// TwinCAT 3 PLC project SlaveController
// ProgramVersion: 3.1.4024.0
// libraries:
//   CAA Memory, * (CAA Technical Workgroup)
//   Tc2_EtherCAT, * (Beckhoff Automation GmbH)
//   Tc2_Math, * (Beckhoff Automation GmbH)
//   Tc2_Standard, * (Beckhoff Automation GmbH)
//   Tc2_System, * (Beckhoff Automation GmbH)
//   Tc2_TcpIp, * (Beckhoff Automation GmbH)
//   Tc2_Utilities, * (Beckhoff Automation GmbH)
//   Tc3_Module, * (Beckhoff Automation GmbH)
// project tree:
//   AgiMaths/Frames/ DHTrans.TcPOU (not stored), invFrame.TcPOU (not stored), rotX.TcPOU (not stored), rotY.TcPOU (not stored), rotZ.TcPOU (not stored), transform.TcPOU (not stored)
//   AgiMaths/MatrixLib/ angAxis2Rot.TcPOU (not stored), cross.TcPOU (not stored), Det5.TcPOU (not stored), Det6.TcPOU (not stored), Det7.TcPOU (not stored), invMat6.TcPOU (not stored), invMat6Old.TcPOU (not stored), invMat3.TcPOU (not stored), invMat7.TcPOU (not stored), Mat3T.TcPOU (not stored), matAdd.TcPOU (not stored), matMultiNum.TcPOU (not stored), matMultiply.TcPOU (not stored), matMultiVec.TcPOU (not stored), matSelfAdd.TcPOU (not stored), vecSelfAdd.TcPOU (not stored), matSelfSub.TcPOU (not stored), matSub.TcPOU (not stored), matTranspose.TcPOU (not stored), rot2AngAxis.TcPOU (not stored), vecAdd.TcPOU (not stored), norm.TcPOU (not stored), normalize.TcPOU (not stored), vecSelfMultiNum.TcPOU (not stored), vecMultiNum.TcPOU (not stored), vecSelfSub.TcPOU (not stored), vecSub.TcPOU (not stored)
//   AgiMaths/ sign.TcPOU (not stored), addVec7.TcPOU (not stored), atan2.TcPOU (not stored), cot.TcPOU (not stored)
//   DUTs/ Account.TcDUT
//   DUTs/Enum/ E_ArmLightCtrlWord.TcDUT (not stored), E_CartJointState.TcTLEO (not stored), E_DriverCtrlWord.TcDUT (not stored), E_DriverOPMode.TcDUT (not stored), E_DriverStatusWord.TcDUT (not stored), E_EndoscopePosture.TcDUT (not stored), E_EndoscopeType.TcDUT (not stored), E_InstrumentType.TcDUT, E_MasterArmState.TcDUT (not stored), E_MatchedSlaveArmIdx.TcDUT (not stored), E_SetupArmState.TcDUT (not stored), E_SlaveArmState.TcDUT
//   DUTs/Structure/MasterSlaveCommunication/ ST_MasterStatus.TcDUT (not stored), ST_SlaveStatus.TcDUT
//   DUTs/Structure/ ST_CartInputDataPool.TcDUT (not stored), ST_EtherCATState.TcDUT, ST_Frame.TcDUT (not stored), ST_InstruOnChipData.TcDUT, ST_InstruStatus.TcDUT (not stored), ST_InstruTypeInfo.TcDUT (not stored), ST_SetupArmCtrlCmds.TcDUT (not stored), ST_SetupInputDataPool.TcDUT (not stored), ST_SlaveArmCtrlCmds.TcDUT, ST_SlaveInputDataPool.TcDUT
//   DUTs/Structure/TasksCommunication/ ST_CartJointData.TcDUT (not stored), ST_CartMotorInput.TcDUT (not stored), ST_CartMotorOutput.TcDUT (not stored), ST_CartStatus.TcDUT (not stored), ST_CartUIData.TcDUT (not stored), ST_MasterJointData.TcDUT (not stored), ST_MotorInputs.TcDUT (not stored), ST_MotorOutputs.TcDUT (not stored), ST_SafetyData.TcDUT, ST_SetupJointData.TcDUT (not stored), ST_SetupStatus.TcDUT, ST_SlaveDynaData.TcDUT (not stored), ST_SlaveJointData.TcDUT (not stored), ST_SlaveUIData.TcDUT (not stored)
//   DUTs/Structure/UICommunication/ ST_cartOperation.TcDUT, ST_instruInfomation.TcDUT, ST_robotStateMachine.TcDUT, ST_uiControl.TcDUT
//   DUTs/Type/ Mat34.TcDUT (not stored), Mat35.TcDUT (not stored), Mat37.TcDUT (not stored), Mat3d.TcDUT (not stored), Mat43.TcDUT (not stored), Mat45.TcDUT, Mat4d.TcDUT (not stored), Mat53.TcDUT (not stored), Mat5d.TcDUT (not stored), Mat67.TcDUT (not stored), Mat6d.TcDUT (not stored), Mat76.TcDUT (not stored), Mat7d.TcDUT (not stored), Vec13d.TcDUT, Vec13di.TcDUT, Vec2i.TcDUT (not stored), Vec3i.TcDUT, Vec3d.TcDUT (not stored), Vec4b.TcDUT (not stored), Vec4d.TcDUT (not stored), Vec4i.TcDUT (not stored), Vec5b.TcDUT (not stored), Vec5d.TcDUT (not stored), Vec5i.TcDUT (not stored), Vec6d.TcDUT (not stored), Vec6i.TcDUT (not stored), Vec7d.TcDUT (not stored), Vec7i.TcDUT (not stored), Vec8b.TcDUT, Vec8d.TcDUT (not stored), Vec8di.TcDUT, Vec8i.TcDUT (not stored)
//   FBs_Auxiliary/ FB_cartJntDisenableDetect.TcPOU (not stored), FB_cartJntEnableDetect.TcPOU (not stored), FB_initMotorPID.TcPOU, FB_InstruNearDetect.TcPOU (not stored), FB_IOCheck.TcPOU (not stored), FB_IOToggleCheck.TcPOU (not stored), FB_rotaButtonDetect.TcPOU (not stored), FB_setupAdjustDetect.TcPOU (not stored), FB_setupJnt5AdjustDetect.TcPOU (not stored), FB_masterConnectionCheck.TcPOU (not stored), FB_Timer.TcPOU, FB_trocarDetect.TcPOU (not stored), FB_PanelDetect.TcPOU, FB_InstrumentDetect.TcPOU, FB_AdjustDetect.TcPOU (not stored)
//   FBs_BasicControllers/ FB_dither.TcPOU (not stored), FB_BasicInstruControl.TcPOU, FBMacroJntControl.TcPOU (not stored), FB_UltrosonicKnifeControl.TcPOU, FB_PID.TcPOU (not stored)
//   FBs_Robots/ FB_Instrument.TcPOU, FB_JointBase.TcPOU (not stored), FB_SlaveCart.TcPOU (not stored), FB_SlaveJoint.TcPOU, FB_SlaveArm.TcPOU, FB_SlaveRobot.TcPOU
//   FBs_SlaveControllers/ FB_SlaveCtrlDisable.TcPOU (not stored), FB_SlaveCtrlInstruCali.TcPOU, FB_SlaveCtrlInstruInvasion.TcPOU (not stored), FB_SlaveCtrlInstruEndoscopeTest.TcPOU, FB_SlaveCtrlInstruRetract.TcPOU (not stored), FB_SlaveCtrlInstruManualTest.TcPOU, FB_SlaveCtrlMountInstru.TcPOU, FB_SlaveCtrlPerformance.TcPOU (not stored), FB_SlaveCtrlPowerBoxCalibration.TcPOU, FB_SlaveCtrlScopeToggle.TcPOU (not stored), FB_SlaveCtrlStop.TcPOU, FB_SlaveCtrlTest.TcPOU, FB_SlaveCtrlPackage.TcPOU (not stored), FB_SlaveCtrlEndoscope.TcPOU (not stored), FB_SlaveCtrlCart.TcPOU (not stored), FB_SlaveCtrlScopeReady.TcPOU (not stored), FB_SlaveCtrlSelfCheck.TcPOU (not stored), FB_SlaveCtrlError.TcPOU, FB_SlaveCtrlInstruReady.TcPOU (not stored), FB_SlaveCtrlMasterSlave.TcPOU, FB_SlaveCtrlAdjust.TcPOU, FB_SlaveCtrlMountPanel.TcPOU, FB_SlaveCtrlPanelReady.TcPOU (unreadable), FB_SlaveCtrlGraCali.TcPOU (not stored), FB_SlaveCtrlInstruAutoTest.TcPOU, FB_SlaveCtrlInstruVerify.TcPOU, FB_SlaveCtrlFrictionTest.TcPOU, FB_SlaveCtrMotorGoHome.TcPOU, FB_SlaveCtrlInit.TcPOU, FB_SlaveCtrlStandBy.TcPOU (unreadable), FB_SlaveArmCtrlBase.TcPOU, I_SlaveArmCtrl.TcIO (not stored)
//   FBs_TrajectoryPlanning/ FB_BasicDoubleS.TcPOU (not stored), FB_trajBase.TcPOU (not stored), FB_TrajMoveJ.TcPOU (not stored), FB_setupTrajMoveJ.TcPOU (not stored), linear_trajectory_with_quintic_polynomial_blends.TcPOU (not stored), quintic_spline_curve.TcPOU (not stored), Quintic_spline_curve_factor.TcPOU (not stored), TrapezoIDal_velocity_trajectory.TcPOU (not stored)
//   FBs_TrajectoryPlanning/OTG/ FB_secOrdTrajFilter.TcPOU (not stored), FB_thirdOrdTrajFilter.TcPOU (not stored)
//   FBs_Filters/ FB_LowPassFilter.TcPOU (not stored)
//   GVLs/ GVL_InstruTestUIVars.TcGVL, GVL_MathDefine.TcGVL, GVL_MES.TcGVL, GVL_SafetyParameters.TcGVL (not stored), GVL_SystemParameters.TcGVL
//   GVLs/Instrument/ GVL_InstruCtrlParams.TcGVL, GVL_InstruTypeDefine.TcGVL
//   GVLs/SlaveArms/ GVL_SlaveArmDynamics.TcGVL, GVL_SlaveArmKinematic.TcGVL (not stored), GVL_SlaveControlParameters.TcGVL, GVL_SlaveJointEncoderCaliData.TcGVL, GVL_SlaveMotorParameters.TcGVL
//   Mains/ SlaveArmControl.TcPOU
//   / RecipeManager.TcRMO (not stored), TaskSlaveArmControl.TcTTO (not stored)
//   SafetyCheck/ ASSERT.TcPOU (not stored), FB_CartCheck.TcPOU (not stored), Fb_ErrRecord.TcPOU (not stored), FB_EtherCATCheck.TcPOU (not stored), Fb_SafetyCheck.TcPOU (not stored), FB_SetupArmCheck.TcPOU (not stored), FB_SlaveArmCheck.TcPOU (not stored), FB_Writer.TcPOU (not stored)
//   SafetyCheck/ErrRecord/ CarErrInputVariable.TcDUT (not stored), checkDelay.TcDUT (not stored), checkDelayTime.TcDUT (not stored), checkInputVariable.TcDUT (not stored), checkPermit.TcDUT (not stored), monitorThreshold.TcDUT (not stored), monitorThreshold_1.TcDUT (not stored), PromptMessage.TcDUT (not stored), ST_Buffer.TcDUT (not stored), T_Buffer.TcDUT (not stored)
//   Sandbox/ FB_SlaveCtrlInstruAutoTest_bak.TcPOU, FB_SlaveCtrlInstruVerify_bak.TcPOU, FB_SlaveCtrlMasterSlave_backup.TcPOU
// real-time tasks:
//   TASK TaskSlaveArmControl: cycle T#250us, priority 1, ADS port 350
// I/O:
//   DEVICE Device 3 (EtherCAT), AmsNetId 192.168.2.195.4.1
//     Box 1 (AX58200_MotorControl) [AX58200_MotorControl_V1001]
//     Box 2 (AX58200_MotorControl) [AX58200_MotorControl_V1001]
// variable links:
//   SlaveController/SlaveController Instance <-> Device 3 (EtherCAT)/Box 1 (AX58200_MotorControl)
//     TaskSlaveArmControl Inputs/SlaveArmControl.m_slaveRobot.m_slaveArms[1].m_joints[4].m_motorInputs/m_current <-> TxPdoMappingCsv/Torque actual value for axis2
//     TaskSlaveArmControl Inputs/SlaveArmControl.m_slaveRobot.m_slaveArms[1].m_joints[5].m_motorInputs/m_current <-> TxPdoMappingCsv/Torque actual value for axis3
//     TaskSlaveArmControl Inputs/SlaveArmControl.m_slaveRobot.m_slaveArms[1].m_joints[4].m_motorInputs/m_linkEncoder <-> TxPdoMappingCsv/ENC for axis2
//     TaskSlaveArmControl Inputs/SlaveArmControl.m_slaveRobot.m_slaveArms[1].m_joints[5].m_motorInputs/m_linkEncoder <-> TxPdoMappingCsv/ENC for axis3
//     TaskSlaveArmControl Inputs/SlaveArmControl.m_slaveRobot.m_slaveArms[1].m_joints[4].m_motorInputs/m_motorEncoder <-> TxPdoMappingCsv/Position actual value for axis2
//     TaskSlaveArmControl Inputs/SlaveArmControl.m_slaveRobot.m_slaveArms[1].m_joints[5].m_motorInputs/m_motorEncoder <-> TxPdoMappingCsv/Position actual value for axis3
//     TaskSlaveArmControl Inputs/SlaveArmControl.m_slaveRobot.m_slaveArms[1].m_joints[4].m_motorInputs/m_statusWord <-> TxPdoMappingCsv/Statusword
//     TaskSlaveArmControl Inputs/SlaveArmControl.m_slaveRobot.m_slaveArms[1].m_joints[5].m_motorInputs/m_statusWord <-> TxPdoMappingCsv/Statusword
//     TaskSlaveArmControl Inputs/SlaveArmControl.m_slaveRobot.m_slaveArms[1].m_panelInstrumentOnIO <-> TxPdoMappingCsv/Digital input
//     TaskSlaveArmControl Outputs/SlaveArmControl.m_slaveRobot.m_slaveArms[1].m_joints[4].m_motorOutputs/m_cmdCurrent <-> RxPdoMappingCsv/Target torque for axis2
//     TaskSlaveArmControl Outputs/SlaveArmControl.m_slaveRobot.m_slaveArms[1].m_joints[5].m_motorOutputs/m_cmdCurrent <-> RxPdoMappingCsv/Target torque for axis3
//     TaskSlaveArmControl Outputs/SlaveArmControl.m_slaveRobot.m_slaveArms[1].m_joints[4].m_motorOutputs/m_cmdMotorEncoder <-> RxPdoMappingCsv/Target position for axis2
//     TaskSlaveArmControl Outputs/SlaveArmControl.m_slaveRobot.m_slaveArms[1].m_joints[5].m_motorOutputs/m_cmdMotorEncoder <-> RxPdoMappingCsv/Target position for axis3
//     TaskSlaveArmControl Outputs/SlaveArmControl.m_slaveRobot.m_slaveArms[1].m_joints[4].m_motorOutputs/m_controlWord <-> RxPdoMappingCsv/Controlword
//     TaskSlaveArmControl Outputs/SlaveArmControl.m_slaveRobot.m_slaveArms[1].m_joints[4].m_motorOutputs/m_opMode <-> RxPdoMappingCsv/Modes of operation
//   SlaveController/SlaveController Instance <-> Device 3 (EtherCAT)/Box 2 (AX58200_MotorControl)
//     TaskSlaveArmControl Inputs/SlaveArmControl.m_slaveRobot.m_slaveArms[1].m_joints[6].m_motorInputs/m_current <-> TxPdoMappingCsv/Torque actual value for axis2
//     TaskSlaveArmControl Inputs/SlaveArmControl.m_slaveRobot.m_slaveArms[1].m_joints[7].m_motorInputs/m_current <-> TxPdoMappingCsv/Torque actual value for axis3
//     TaskSlaveArmControl Inputs/SlaveArmControl.m_slaveRobot.m_slaveArms[1].m_joints[6].m_motorInputs/m_linkEncoder <-> TxPdoMappingCsv/ENC for axis2
//     TaskSlaveArmControl Inputs/SlaveArmControl.m_slaveRobot.m_slaveArms[1].m_joints[7].m_motorInputs/m_linkEncoder <-> TxPdoMappingCsv/ENC for axis3
//     TaskSlaveArmControl Inputs/SlaveArmControl.m_slaveRobot.m_slaveArms[1].m_joints[6].m_motorInputs/m_motorEncoder <-> TxPdoMappingCsv/Position actual value for axis2
//     TaskSlaveArmControl Inputs/SlaveArmControl.m_slaveRobot.m_slaveArms[1].m_joints[7].m_motorInputs/m_motorEncoder <-> TxPdoMappingCsv/Position actual value for axis3
//     TaskSlaveArmControl Inputs/SlaveArmControl.m_slaveRobot.m_slaveArms[1].m_joints[6].m_motorInputs/m_statusWord <-> TxPdoMappingCsv/Statusword
//     TaskSlaveArmControl Inputs/SlaveArmControl.m_slaveRobot.m_slaveArms[1].m_joints[7].m_motorInputs/m_statusWord <-> TxPdoMappingCsv/Statusword
//     TaskSlaveArmControl Inputs/SlaveArmControl.m_slaveRobot.m_slaveArms[1].m_joints[8].m_motorInputs/m_statusWord <-> TxPdoMappingCsv/Statusword
//     TaskSlaveArmControl Inputs/SlaveArmControl.m_slaveRobot.m_slaveArms[1].m_joints[8].m_motorInputs/m_current <-> TxPdoMappingCsv/Torque actual value
//     TaskSlaveArmControl Inputs/SlaveArmControl.m_slaveRobot.m_slaveArms[1].m_joints[8].m_motorInputs/m_linkEncoder <-> TxPdoMappingCsv/ENC
//     TaskSlaveArmControl Inputs/SlaveArmControl.m_slaveRobot.m_slaveArms[1].m_joints[8].m_motorInputs/m_motorEncoder <-> TxPdoMappingCsv/Position actual value
//     TaskSlaveArmControl Outputs/SlaveArmControl.m_slaveRobot.m_slaveArms[1].m_joints[6].m_motorOutputs/m_cmdCurrent <-> RxPdoMappingCsv/Target torque for axis2
//     TaskSlaveArmControl Outputs/SlaveArmControl.m_slaveRobot.m_slaveArms[1].m_joints[7].m_motorOutputs/m_cmdCurrent <-> RxPdoMappingCsv/Target torque for axis3
//     TaskSlaveArmControl Outputs/SlaveArmControl.m_slaveRobot.m_slaveArms[1].m_joints[6].m_motorOutputs/m_cmdMotorEncoder <-> RxPdoMappingCsv/Target position for axis2
//     TaskSlaveArmControl Outputs/SlaveArmControl.m_slaveRobot.m_slaveArms[1].m_joints[7].m_motorOutputs/m_cmdMotorEncoder <-> RxPdoMappingCsv/Target position for axis3
//     TaskSlaveArmControl Outputs/SlaveArmControl.m_slaveRobot.m_slaveArms[1].m_joints[6].m_motorOutputs/m_controlWord <-> RxPdoMappingCsv/Controlword
//     TaskSlaveArmControl Outputs/SlaveArmControl.m_slaveRobot.m_slaveArms[1].m_joints[6].m_motorOutputs/m_opMode <-> RxPdoMappingCsv/Modes of operation
//     TaskSlaveArmControl Outputs/SlaveArmControl.m_slaveRobot.m_slaveArms[1].m_joints[8].m_motorOutputs/m_cmdCurrent <-> RxPdoMappingCsv/Target torque
//     TaskSlaveArmControl Outputs/SlaveArmControl.m_slaveRobot.m_slaveArms[1].m_joints[8].m_motorOutputs/m_cmdMotorEncoder <-> RxPdoMappingCsv/Target position

// ---- DUTs/Account.TcDUT
TYPE Account :
STRUCT
	logOn:BOOL;
	logOut:BOOL;
	autoLogOut:BOOL;
	register:BOOL;//注册
	actualAccountNumber:STRING;
	actualPassWord:STRING;
	actualPermission:USINT;//权限 0 无登录 1 管理 2 研发 3 质量 4 生产
	actualWorkNum:UDINT;
	actualName:STRING;
	registerAccountNumber:STRING;
	registerPassWord:STRING;
	registerPermission:USINT;
	registerWorkNum:UDINT;
	registerName:STRING;
	prompt:STRING;//提示
	memoryAccountNumber:ARRAY [0..50] OF STRING; //注册账号
	memoryPassWord:ARRAY [0..50] OF STRING; //注册账密码
	memoryPermission:ARRAY [0..50] OF USINT; //注册账权限
	memoryWorkNum:ARRAY [0..50] OF UDINT;//注册账工号
	memoryName:ARRAY [0..50] OF STRING; //注册账姓名
	memoryTime:ARRAY [0..50] OF STRING; //注册时间
	memoryDisable:ARRAY [0..50] OF BOOL;//使能
END_STRUCT
END_TYPE

// ---- DUTs/Enum/E_InstrumentType.TcDUT
TYPE E_InstrumentType :
(
	InstruType_UNKNOWM := 0,
	InstruType_CadiereForceps :=7,
	InstruType_NeedleDriver :=8,
	InstruType_MegaSCNeedleDriver :=9,// mega suture-cut needle driver
	InstruType_SCNeedleDriver :=10, // suture-cut needle driver
	InstruType_RoundTipScissors :=11,
	InstruType_ProGraspForceps :=12,
	InstruType_MarylandForceps :=13, // Maryland bipolar forceps
	InstruType_FenestratedForceps :=14, // Fnestrated bipolar forceps
	InstruType_CurvedScissors :=15, // monopolar curved scissors
	InstruType_CauteryHook :=16,
	InstruType_CauterySpatula :=17,
	InstruType_Endoscope := 20,
	InstruType_NewEndoscope := 31,
	InstruType_UltrasoundKnifeS :=42,
	InstruType_UltrasoundKnifeU :=43,
	InstruType_TipUpFenestratedGrasper :=44,
	InstruType_MegaNeedleDriver :=45,
	InstruType_DeBakeyForceps :=46,
	InstruType_BlackDiamondForceps :=47,
	InstruType_PottsScissors :=48,
	InstruType_CurvedBipolarDissector :=49,
	InstruType_MicroBipolarForceps :=50,
	InstruType_ForceBipolar :=51,
	InstruType_MicroCauteryHook :=52,
	InstruType_CENewEndoscope := 320
);
END_TYPE

// ---- DUTs/Enum/E_SlaveArmState.TcDUT
TYPE E_SlaveArmState :
(
	SlaveArmState_Error := 1,
	SlaveArmState_Init :=2,
	SlaveArmState_SelfCheck :=3,
	SlaveArmState_Standby :=4,
	SlaveArmState_MountPanel:=5,
	SlaveArmState_PanelReady :=6,
	SlaveArmState_MountInstru :=7,
	SlaveArmState_InstruReady :=8,
	SlaveArmState_MasterSlave :=9,
	SlaveArmState_ScopeReady :=10,
	SlaveArmState_EndoScope :=11,
	SlaveArmState_Adjust :=12,
	SlaveArmState_Package :=13,
	SlaveArmState_Cart := 14,
	SlaveArmState_GravityCali := 15,
	SlaveArmState_Test := 16,
	SlaveArmState_InstruRetract :=17,
	SlaveArmState_InstruInvasion :=18,
	SlaveArmState_Disable := 19,
	SlaveArmState_InstruCali := 20,
	SlaveArmState_ScopeToggle :=21,
	SlaveArmState_Performance:=22,
	SlaveArmState_Stop :=23,
	SlaveArmState_InstruAutoTest :=24,
	SlaveArmState_InstruManualTest :=25,
	SlaveArmState_InstruVerify :=26,
	SlaveArmState_MotorGoHome:= 27,
	SlaveArmState_PowerBoxCalibration:= 28,
	SlaveArmState_EndoscopeTest:= 29,
	SlaveArmState_FrictionTest:= 30,
	
	SlaveArmState_Jnt5Rotate:=31,
	SlaveArmState_totalNum :=SlaveArmState_Jnt5Rotate
);
END_TYPE

// ---- DUTs/Structure/MasterSlaveCommunication/ST_SlaveStatus.TcDUT
// Output from slave arm control task, including arm status and cartesian data
// Input to safety task and Master controller
TYPE ST_SlaveStatus :
STRUCT
	
	// state machine
	m_armState:ARRAY[1..g_sArmNum] OF E_SlaveArmState:=[g_sArmNum(SlaveArmState_Error)];
	
	// self-check pass flag
	m_selfCheckPass :ARRAY[1..g_sArmNum] OF BOOL :=[g_sArmNum(False)];
	
	// instrument info
	m_instruStauts :ARRAY[1..g_sArmNum] OF ST_InstruStatus;
	
	// flag if endoscope is mounted
	m_endoscopeMounted :BOOL := FALSE;
	
	// endoscope pose in cart coordinate
	m_endoscopePose : ST_Frame;
	
	// command arm pose in slave arm coordinate
	m_cmdArmPose:ARRAY[1..g_sArmNum] OF ST_Frame;
	
	// current arm pose in slave arm coordinate
	m_curArmPose:ARRAY[1..g_sArmNum] OF ST_Frame;
	
	// simulation arm pose in slave arm coordinate
	m_simArmPose:ARRAY[1..g_sArmNum] OF ST_Frame;
	
	// master slave pose error [position, angle*axis] in endoscope coordinate
	m_masterSlavePoseError :ARRAY[1..g_sArmNum] OF Vec6d; 

	//read instrument information error ID
	m_instruReadErrId : ARRAY[1..g_sArmNum] OF INT;
	
	//instrument install status
	m_instruInstallStatus : ARRAY[1..g_sArmNum] OF BOOL;
	
	//instrument clamp error Id 
	m_instruClampErrId : ARRAY[1..g_sArmNum] OF UINT;
	
	//panel install status
	m_panelInstallStatus : ARRAY[1..g_sArmNum] OF BOOL;
	
	//panel clamp error ID
	m_panelClampErrId : ARRAY[1..g_sArmNum] OF UINT;
	
	//trocar install status 
	m_trocarOnFlag : ARRAY[1..g_sArmNum] OF BOOL;

	// flag if master are connected
	m_masterOnLine :BOOL ;
	
	// slave robot stop button trigger 
	m_slaveStopButton : BOOL;
END_STRUCT
END_TYPE

// ---- DUTs/Structure/ST_EtherCATState.TcDUT
TYPE ST_EtherCATState :
STRUCT
	EtherCATState : BOOL;
	CRCPortA :UDINT;
	CRCPortB :UDINT;
	CRCPortC :UDINT;
END_STRUCT
END_TYPE

// ---- DUTs/Structure/ST_InstruOnChipData.TcDUT
TYPE ST_InstruOnChipData :
STRUCT

	// ID
	m_InstruID: INT:=0;
	
	// series number
	m_InstruseriesNum : ULINT:=0;
	
	// current and max usage counts
	m_InstruUsageCounts :ULINT;
	m_InstrumaxUsageCounts :ULINT:=20;
	
	//Instrument Zero augular offset
	m_InstruPos:Vec5d;
	//Instrument RFID 
	m_InstruPosRFID:Vec5d;
	m_InstruIDFromRFID: INT:=0;
	m_InstruUsageCountsRFID :ULINT;
	m_InstruReadSucceedRFID:BOOL;
	m_InstruseriesNumRFID : ULINT:=0;
	//Instrument state
	m_InstruReadSucceed:BOOL;
	
	//Instrument Clamp Error
	m_Error:BOOL;
	m_ErrorID:INT;//1器械类型错误、2器械使用次数超限、3两个内窥镜
	
	m_InstruPurpose :ULINT;
	m_InstruPurposeTime :ULINT;
END_STRUCT
END_TYPE

// ---- DUTs/Structure/ST_SlaveArmCtrlCmds.TcDUT
TYPE ST_SlaveArmCtrlCmds :
STRUCT
	// arm control data
	// NOTE: simulated joint position is usd for kinematic controller 
	//		while command joint position is used for real robot controller
	// 		They are identical for the most time, but in some cases, simulated position is filted to get command one 
	m_jntEnableFlag : Vec8i;
	m_jntOPMode : Vec8i;
	m_simJntPos : Vec8d;
	m_cmdJntPos : VEC8d;
	m_cmdJntVel : VEC8d;
	m_cmdJntAcc : VEC8d:=g_zeroVec8d;
	m_cmdJntTrq : VEC8d:=g_zeroVec8d;
	m_cmdCartPose : ST_Frame;
	m_cmdCartTwist : Vec6d;
	m_FFJntTrq :Vec8d:=g_zeroVec8d;
	
END_STRUCT
END_TYPE

// ---- DUTs/Structure/ST_SlaveInputDataPool.TcDUT
// Struct contains all data from other tasks and controller used for slave control
TYPE ST_SlaveInputDataPool :
STRUCT
		
	// UI information, import from UI controller
	m_UIData :ST_SlaveUIData;
	
	// safety information, import from safety check task
	m_safetyData : ST_SafetyData;
	
	// cart information, import from other task
	m_cartStatus :ST_CartStatus;
	
	// master robot status, copy from MSCommu_MasterStatus
	m_masterStatus :ST_MasterStatus;
	
	// setup arms infromation;
	m_setupStatus : ST_SetupStatus;
	
	// slave dynamic data
	m_slaveDynaData : ST_SlaveDynaData;
	
END_STRUCT
END_TYPE

// ---- DUTs/Structure/TasksCommunication/ST_SafetyData.TcDUT
// Output from safety check task
// Input to master arm control task
TYPE ST_SafetyData :
STRUCT
	m_slaveErrFlag :ARRAY[1..g_sArmNum] OF BOOL :=[g_sArmNum(FALSE)];
	m_setupErrFlag :ARRAY[1..g_sArmNum] OF BOOL :=[g_sArmNum(FALSE)];
	m_cartErrFlag :BOOL :=FALSE;
	m_cartSteadyFootErr :BOOL;
	m_cartWheelErr :BOOL;
	m_cartStandColumnErr :BOOL;
	m_cartAdjustErr :BOOL;
	m_cartOverhangErr :BOOL;
END_STRUCT
END_TYPE

// ---- DUTs/Structure/TasksCommunication/ST_SetupStatus.TcDUT
TYPE ST_SetupStatus :
STRUCT
	// state machine
	m_armState:ARRAY[1..g_sArmNum] OF E_SetupArmState:=[g_sArmNum(SetupArmState_Error)];
	
	// current pose of set arm distal end
	m_curEndPose:ARRAY[1..g_sArmNum] OF ST_Frame;
	
	// position of remote center point
	m_rcPos :ARRAY[1..g_sArmNum] OF Vec3d;
END_STRUCT
END_TYPE

// ---- DUTs/Structure/UICommunication/ST_cartOperation.TcDUT
TYPE ST_cartOperation :
STRUCT
	//sterile state ,  0 : unfinshed  , 1 : complete
	m_setupSterileStateArm1 : UINT;
	m_setupSterileStateArm2 : UINT;
	m_setupSterileStateArm3 : UINT;
	m_setupSterileStateArm4 : UINT;
	
	//draping adjust state , 0 : unfinshed  , 1 : finshed
	m_drapingAdjustState : UINT;

	//sterile install state , 0 : unfinshed  , 1 : finshed
	m_setupSterileState : UINT;

	//docking adjust state , 0 : unfinshed  , 1 : finshed
	m_dockingAdjustState : UINT;
	
	//cart in the sterile area 
	m_cartInSterileState : UINT;
	
	//scope installed , 0 : unfinshed  , 1 : finshed
	m_scopeInstalled :UINT;
	
	//robot in surgical allowed , scope installed and an arm mounted instrument
	m_inSurgicalAllowed : UINT;
	
	//arm storage completed
	m_armStorageCompleted : UINT;
END_STRUCT
END_TYPE

// ---- DUTs/Structure/UICommunication/ST_instruInfomation.TcDUT
TYPE ST_instruInfomation :
STRUCT
	//instrument is ready
	m_instruIsConnected : BOOL;
	
	//new instrument  true
	m_newInstrument : BOOL;
	
	//instrument arm in master-slave
	m_instruInMasterSlave : BOOL;
	
	//master send  pedal active
	m_pedalHover : BOOL;
	
	//0 : Passive instrument , 1 : unipolar instrument , 2 : bipolar instrument, 3 : ultrasound knife, 4 : endoscope
	m_instruType : UINT;
	
	//master send  pedal hover
	m_pedalActive : UINT;
	
	//arm id
	m_armId : UINT;
	m_instruID : UINT;
	
	//instrument total number
	m_instruTotalLife : UINT := 100;
	
	//instrument use life (ui write)
	m_useLifeUi : UINT;

	//instrument  use life (plc write)
	m_useLifeplc : UINT;
	
	//instrument serial number
	m_instruSerialNum : LINT;
	
	m_instruPosX : REAL;
	m_instruPosY : REAL;
	m_instruPosZ : REAL;

	//instrument English name 
	m_nameEn : STRING;
	
	//instrument Chinese name 
	m_nameCh : WSTRING;
	
END_STRUCT
END_TYPE

// ---- DUTs/Structure/UICommunication/ST_robotStateMachine.TcDUT
TYPE ST_robotStateMachine :
STRUCT
	m_stateMachineCart : INT;
	m_stateMachineArm1 : INT;
	m_stateMachineArm2 : INT;
	m_stateMachineArm3 : INT;
	m_stateMachineArm4 : INT;

END_STRUCT
END_TYPE

// ---- DUTs/Structure/UICommunication/ST_uiControl.TcDUT
TYPE ST_uiControl :
STRUCT
	//台车自动摆位---姿态调整为建立无菌屏障时所需状态--结束后给定结束信号
	m_drapingEnable : BOOL;
	
	//台车自动摆位---姿态调整为进入无菌区时所需状态（器械对接姿态）--结束后给定结束信号
	m_dockingEnable : BOOL;
	
	//所有机械臂收纳使能
	m_packageEnable : BOOL;
	
	//通过手柄按钮，任意拖动机械臂所有关节
	m_joystickEnable : BOOL;
	
	//相机界面中的使能按钮
	m_cameraJoystickEnable : BOOL;
	
	 //限制高度调整，true:使能，false:禁止
	m_heightLimitAdjustEnable : BOOL;
END_STRUCT
END_TYPE

// ---- DUTs/Type/Mat45.TcDUT
TYPE Mat45 : ARRAY[1..4, 1..5] OF LREAL; END_TYPE

// ---- DUTs/Type/Vec13d.TcDUT
TYPE Vec13d : ARRAY[1..13] OF LREAL; END_TYPE

// ---- DUTs/Type/Vec13di.TcDUT
TYPE Vec13di : ARRAY[1..13] OF DINT; END_TYPE

// ---- DUTs/Type/Vec3i.TcDUT
TYPE Vec3i : ARRAY[1..3] OF INT; END_TYPE

// ---- DUTs/Type/Vec8b.TcDUT
TYPE Vec8b : ARRAY[1..8] OF BOOl; END_TYPE

// ---- DUTs/Type/Vec8di.TcDUT
TYPE Vec8di : ARRAY[1..8] OF DINT; END_TYPE

// ---- GVLs/GVL_InstruTestUIVars.TcGVL
{attribute 'qualified_only'}
VAR_GLOBAL
	//################ input variables from HMI ########################
	// control variable for instrument calibration
	g_instruCaliFlag :BOOL:= FALSE; // 允许标定按键，按下不反弹
	g_searchZeroPosFlag :BOOL := FALSE; // 器械找零点按键， 按下反弹
	g_writeZeroPosFlag :BOOL :=FALSE; // 器械零位写入，按下反弹
	g_newInstruSN :STRING; // 新序列号
	g_writeSNFlag :BOOL := FALSE; // 新序列号写入， 按下反弹
	
	// control variable for instrument auto test
	g_instruAutoTestFlag :BOOL :=FALSE; // 器械自动测试按键，按下不反弹
	g_instruAutoTestMode :INT :=0; //  自动测试模式 0: 器械开合 1: 器械开合加运动 ; 2: 器械加紧运动
	g_maxInstruAutoTestCycles :DINT :=0; // 最大测试次数
	g_autoTestCycles :INT :=0;
	// control variable for instrument manual test
	g_instruManualTestFlag :BOOL :=FALSE; // 器械手动测试按键，按下不反弹
	g_moveToSetPosFlag :BOOL :=FALSE; // 运动到指令位置 ，按下反弹
	g_targetRollAng :LREAL :=0; //器械回转角度
	g_targetPitchAng :LREAL :=0;//器械俯仰角度
	g_targetYawAng :LREAL :=0;//器械偏摆角度
	g_targetGripAng :LREAL :=0;//器械张开角度
	g_targetGripForceLevel:INT :=0; // 器械夹持力百分比
	g_gripperOpenFlag :BOOL :=FALSE; // 命令器械张开按键, 按下反弹
	g_gripperCloseFlag :BOOL :=FALSE; // 命令器械闭合按键, 按下反弹
	g_maxGripForceFlag :BOOL :=FALSE;// 命令器械最大加紧力按键, 按下反弹
	g_forceBipolarMode : BOOL := FALSE;
	g_forceBipolarModeAllowed : BOOL := FALSE;
	
	// control variable for instrument verify
	g_instruVerifyFlag :BOOL :=FALSE; // 器械验证按键，按下不反弹
	g_instruVerifyLastStepFlag :BOOL:=FALSE; // 下一步按键， 按下反弹
	g_instruVerifyNextStepFlag :BOOL :=FALSE; // 上一步按键，按下反弹
	
	//friction test
	g_instruFrictionTestAllowed : BOOL;
	g_instruFrictionTest : BOOL;
	
	//################ output variables  HMI ########################
	g_curInstruJntPos :Vec5d;   // 当前器械角度位置
	g_curInstruJntCurrent:Vec5d; // 当前关节电流
	g_curInstruDHPos :Vec3d; // DH 角度
	g_curGripAng:LREAL; // 当前张开角度
	g_instruZeroPos :Vec5d; // 当前零位
	g_instruSN :STRING; // 当前序列号
	g_maxGripAng:LREAL:=45; // 当前张开角度
	// 读取器械信息
	g_readInstruInformation: BOOL;
	// 信息校验通过
	g_informationVerificationPassed: BOOL;
	// 电机使能
	g_powerOn: BOOL;
	// 电机使能状态
	g_enabled: BOOL;
	// 卡接隔离板
	g_snappingSeparator: BOOL;
	// 电机停止
	g_motorStops: BOOL;
	// 器械卡接找点
	g_instrumentSnapping: BOOL;
	// 器械自动卡接
	g_instrumentAutoSnapping: BOOL;
	// 器械卡接停止
	g_instrumentSnappingStop: BOOL;
	// 位置写入芯片
	g_positionWritingChip: BOOL;
	// 位置数据写入
	g_writeENC2PosData: LREAL;
	// 读取器械信息状态
	g_readInstruinformationFlag: BOOL;
	// 读取到的SN码
	g_readSNNum: ULINT;
	// 器械使用次数
	g_instruNumberOfUses: UINT;
	// 器械总使用次数
	g_instruNumberOfAllUses: UINT;
	// 增加使用次数
	g_incInstruNumOfUses: BOOL;
	// 清除使用次数
	g_clearInstruNumOfUses: BOOL;
	// 位置从芯片读取
	g_readENC2PosData: BOOL;
	// 写入器械中的SN码
	g_writeSNNum: ULINT;
	// 写入SN码
	g_writeInstruSN: BOOL;
	// 写入器械用途
	g_writeInstruPurpose: BOOL;
	// 写入器械的用途
	g_writePurposeNum: UINT;
	// 修改额定电流
	g_modifyRatedCurrent: BOOL;
	// 目标额定电流
	g_targetRatedCurrent: LREAL;
	// 实际额定电流
	g_actualRatedCurrent: ARRAY[1..g_sJntNum] OF LREAL := [8(800)];
	// 动力盒标定状态
	g_powerBoxCalibrationFlag: BOOL := TRUE;
	// 动力盒标定
	g_powerBoxCalibration: BOOL;
	// 动力盒回零位
	g_goHome: BOOL;
	
	// 读取器械用途
	g_readInstruPurpose: UINT;
	// 读取器械的用途
	g_readPurposeTime: UINT;	
	g_instruNameCN : WSTRING := " ";
	
	// 清除壳体次数
	g_jnt5RotateFlag:BOOL:=FALSE;
END_VAR
VAR_GLOBAL RETAIN PERSISTENT
	// 动力盒零位已校准
	g_powerBoxCalibrationed: BOOL;
	// 动力盒零位
	g_powerBoxCalibrationPos: ARRAY [1..g_sArmNum, 1..g_sJntNum] OF DINT;
	// 账户
	g_account: Account := (memoryAccountNumber := ['admin', 50('')], memoryPassWord := ['yfAGIBOT2025', 50('')], memoryPermission := [1, 50(0)], memoryWorkNum := [1, 50(0)], memoryName := ['admin', 50('')]);
END_VAR
VAR_GLOBAL
	// 动力盒零位状态
	g_beHomed: BOOL;
	// 后台启用角度补偿
	g_enableBackendCompensation: BOOL;
	// 研发启用角度补偿
	g_enableRDCompensation: BOOL;
	// DH补偿角度
	g_compensationAngleDH: Vec3d;
	// DH补偿角度内部
	g_compensationAngleBackendDH: Vec3d;
	// 俯仰
	g_pitchAngularVel: LREAL;
	// 偏摆/开合
	g_deviationAngularVel: LREAL;
	// 旋转
	g_rotationAngularVel: LREAL;
	// 俯仰加速度
	g_pitchAngularAcc: LREAL;
	// 偏摆/开合加速度
	g_deviationAngularAcc: LREAL;
	// 旋转加速度
	g_rotationAngularAcc: LREAL;
	// 俯仰目标电流
	g_pitchTargetCurrent: LREAL;
	// 偏摆/开合目标电流
	g_deviationTargetCurrent: LREAL;
	// 旋转目标电流
	g_rotationTargetCurrent: LREAL;
	// 俯仰当前电流
	g_pitchActualCurrent: LREAL;
	// 偏摆/开合当前电流
	g_deviationActualCurrent: LREAL;
	// 旋转当前电流
	g_rotationActualCurrent: LREAL;
	// 当前状态集
	g_stateMachine: E_SlaveArmState;
	// 循环设定次数
	g_testCycles: INT;
	// 自动测试开始
	g_autoTestStart: BOOL;
	// 自动测试结束
	g_autoTestStop: BOOL;
	// 电流是否到达功能
	g_funcCurrentDetection: BOOL;
	// 测试时间时
	g_testTimeHour: UINT;
	// 测试时间分
	g_testTimeMinute: UINT;
	// 测试时间秒
	g_testTimeSecond: UINT;
	// 测试模式
	g_testMode: INT;
	// 最大开合角
	g_maxGripAngle: LREAL := 45;
	// 自动测试步骤
	g_testStep: INT;
	// 最小开合角
	g_minGripAngle: LREAL:=-45;
	// 在位置
	g_inPos: BOOL;
	// 下一步
	g_nextStep: BOOL;
	// 上一步
	g_lastStep: BOOL;
	// 当前循环次数
	g_curTestCycles: INT;
	// 自动测试暂停
	g_autoTestPause: BOOL;
	// 读取RFID状态
	g_readRFIDFlag: BOOL;
	// 器械标定状态
	g_instruCaliState: BOOL;
	g_jogClose:BOOL;
	
	writeInstruZeroPos :Vec5d; // 当前写入器械零位
	g_clearInformation:BOOL;//清除账户账号信息
	
	g_offLineRFID:BOOL;
//	g_informationVerificationPassed:BOOL;
	g_readedRFID:BOOL;
	g_readRFID:BOOL;
	g_writeRFID:BOOL;
	g_RFID_SN:STRING;
	m_RFIDTimes:DINT;
	m_Instrument_pos_L1:LREAL;
	m_Instrument_pos_L2:LREAL;
	m_Instrument_pos_L3:LREAL;
	m_postureTestStep:INT;
	m_cycleStart: BOOL;
	m_cycleStop: BOOL;
	g_endoscopeAngle: INT;
	g_endoscopeTest: BOOL;
	g_endoscopeUpturnFlagBit: BOOL;
	g_endoscopeUpturn30FlagBit: BOOL;
	g_manualPowerBoxCalibration: BOOL;
	g_writeZeroPosFlagErr:BOOL;
	g_logOutEnable:BOOL;
	g_maxAngleEnable:BOOL;
	g_maxAngle:LREAL;
	g_cycleEndoscopeTest:INT;
	g_startEndoscopeTest:BOOL;
	g_instruSNLen:INT;
	g_snappingSeparatoring:BOOL;
	g_instruAutoSnapping:BOOL;
	g_instruCalibrationing:BOOL;
	g_disableAccount:BOOL;
	g_accountDelete:BOOL;
	g_accountSN:INT;
	g_queryAccountSN:INT;
	g_queryAccountFlag:BOOL;
	g_queryAccountNumber:STRING;
	g_queryPassWord:STRING;
	g_queryPermission:USINT;
	g_queryWorkNum:UDINT;
	g_queryName:STRING;
	g_queryTime:STRING;
	g_queryClear:BOOL;
	g_maxRollEnable:BOOL;
	g_maxRoll:LREAL;
	g_maxPitchEnable:BOOL;
	g_maxPitch:LREAL;
	g_maxYawEnable:BOOL;
	g_maxYaw:LREAL;
	g_standbyEnable:BOOL;
	g_testEnable:BOOL;
END_VAR

// ---- GVLs/GVL_MathDefine.TcGVL
VAR_GLOBAL CONSTANT
	g_smallNum :LREAL := 1E-8;
	g_smallAng :LREAL := 0.0001*PI/180;
	g_largeNum: LREAL :=1E16;
	g_deg2Rad :LREAL := pi/180.0;
	g_rad2Deg :LREAL := 180.0/pi;
	g_2pi :LREAL :=2*PI;
	
	g_eye3d :Mat3d:=[1, 0, 0,
					 0, 1, 0,
					 0, 0, 1];
	g_eye4d :Mat4d:=[1, 0, 0, 0,
					 0, 1, 0, 0,
					 0, 0, 1, 0,
					 0, 0, 0, 1];
	g_zeroMat3d :Mat3d:=[9(0)];
	g_zeroMat35 :Mat35:=[15(0)];
	g_zeroMat6d :Mat6d:=[36(0)];
	g_zeroMat7d :Mat7d:=[49(0)];
	g_eye7d :Mat7d:=[1, 0, 0, 0, 0, 0, 0, 
					 0, 1, 0, 0, 0, 0, 0, 
					 0, 0, 1, 0, 0, 0, 0, 
					 0, 0, 0, 1, 0, 0, 0,
					 0, 0, 0, 0, 1, 0, 0,
					 0, 0, 0, 0, 0, 1, 0,
					 0, 0, 0, 0, 0, 0, 1];
	
	g_zeroVec3d :Vec3d:= [3(0)];
	g_onesVec3d: Vec3d:=[3(1)];
	
	g_zeroVec4b :Vec4b := [4(FALSE)];
	g_zeroVec4d :Vec4d:= [4(0)];
	
	g_zeroVec6d: Vec6d:=[6(0)];
	g_onesVec6d: Vec6d:=[6(1)];
	
	g_zeroVec5d: Vec5d:=[5(0)];
	g_onesVec5d: Vec5d:=[5(1.0)];
	g_zeroVec5i: Vec5i:=[5(0)];
	g_onesVec5i: Vec5i:=[5(1)];
	
	g_zeroVec7d: Vec7d:=[7(0)];
	g_onesVec7d: Vec7d:=[7(1.0)];
	g_zeroVec7i: Vec7i:=[7(0)];
	g_onesVec7i: Vec7i:=[7(1)];
	g_zeroVec8b: Vec8b:=[8(FALSE)];
	g_onesVec8b: Vec8b:=[8(TRUE)];
	g_zeroVec8d: Vec8d:=[8(0)];
	g_onesVec8d: Vec8d:=[8(1.0)];
	g_zeroVec8i: Vec8i:=[8(0)];
	g_onesVec8i: Vec8i:=[8(1)];
	g_initCurVec8d :Vec8d:=[8(250)];
	
	g_setupAllPosMode:Vec5i:=[5(DriverOPMode_Pos)];
	g_setupAllTrqMode:Vec5i:=[5(DriverOPMode_Trq)];
	g_slaveAllPosMode:Vec8i:=[8(DriverOPMode_Pos)];
	g_slaveAllTrqMode:Vec8i:=[8(DriverOPMode_Trq)];
	g_slaveAllPosTrqMode:Vec8i:=[8(DriverOPMode_PosTrq)];
	
	
END_VAR

// ---- GVLs/GVL_MES.TcGVL
{attribute 'qualified_only'}
VAR_GLOBAL
	g_serialNum:STRING;
	g_actualAccountNumber:STRING;
	g_powerBoxCalibrationPos: ARRAY [1..g_sArmNum, 1..g_sJntNum] OF DINT;
	g_SN:STRING;
	g_writeInstruZeroPos :Vec5d; 
	g_instruZeroPos	:Vec5d; 
	g_readRFIDFlig:BOOL;
	g_curNumTiredTest:INT;
	g_attitudeConfirm:INT;
	g_attitudeOK:BOOL;
	g_attitudeNG:BOOL;
	g_eventTime:ARRAY [1..9] OF  STRING;
	g_serialNumLen:INT;
	g_autoTestMode:INT;
END_VAR

// ---- GVLs/GVL_SystemParameters.TcGVL
VAR_GLOBAL CONSTANT
	
	g_InstruTestVersion : WSTRING := "STST01 器械测试平台 V1(1.3.0.1) ";
	g_mArmNum :INT := 2;	
	g_mJntNum :INT := 7;	
	g_sArmNum :INT := 1;	
	g_sJntNum :INT := 8;
	g_setupJntNum :INT :=5;
	g_cartDofs :INT :=6;
	g_cartJntNum:INT :=8;
	
	
	
	// control loop interval for each task
	g_slaveArmCtrlCycleTime :LREAL :=0.00025;
	g_slaveArmCtrlFreq :LREAL :=1.0/g_slaveArmCtrlCycleTime;
	g_armDynamicCycleTime :LREAL := 0.001;
	g_armDynamicFreq :LREAL := 1.0/g_armDynamicCycleTime;
	g_setupArmCtrlCycleTime :LREAL := 0.001;
	g_setupArmCtrlFreq :LREAL := 1.0/g_setupArmCtrlCycleTime;
	g_cartCtrlCycleTime :LREAL := 0.001;
	g_cartCtrlFreq :LREAL := 1.0/g_cartCtrlCycleTime;
	
	// wait time before robot init  for ethercat to stablize 
	g_robotInitWaitTime : LREAL := 1.0;
	RecipeDefinitionName :ARRAY [1..2] OF STRING := ['account', 'caliLinkEncoder'];
END_VAR

// ---- GVLs/Instrument/GVL_InstruCtrlParams.TcGVL
// NOTICE： Use m_instruTypeIdx in FB_Instrument as the array index to get data below
{attribute 'global_init_slot' := '49991'}
VAR_GLOBAL CONSTANT
	// master gripper angle limit
	g_maxMasterGripAngle :LREAL := 30*g_deg2Rad;
	g_minMasterGripAngle : LREAL :=0.0;
	g_masterGripForceStartAng :LREAL :=5*g_deg2Rad;
	
	// gripper angle corresponding to g_masterGripForceStartAng
	// make sure fingers are fully closed and have a initial force
	g_minSlaveGripAngle :LREAL := -20 * g_deg2Rad; 
	
	//ultrasound knife kinematics parameter
	g_uknifeGripTravel :LREAL:= 0.00353;
	g_uknifeGripDividAngle : LREAL := 17 * g_deg2Rad;
	g_uknifeMotorLead : LREAL := 0.025;
	g_uknifeLeverRatio : LREAL := 13.0/18.5;
	
	// prograsp kinematic parameters
	g_proGraspAB :LREAL :=2.8;
	g_proGraspBC :LREAL :=5.26;
	g_proGraspInitA :LREAL :=16.6*g_deg2Rad;;
	g_proGraspInitC :LREAL :=8.75*g_deg2Rad;
	
	g_proGrasp2AB :LREAL :=2.7;
	g_proGrasp2BC :LREAL :=5.254;
	g_proGrasp2InitA :LREAL :=16.13*g_deg2Rad;;
	g_proGrasp2InitC :LREAL :=8.21*g_deg2Rad;
	
	// instrument grip yaw compensation
	g_instruBacklashDir: ARRAY[1..5] OF INT :=[-1, -1, -1, 1, 0];
	g_instruGripYawCompAng :ARRAY[1..4] OF LREAL := [ 2*g_deg2rad,  4*g_deg2rad,  6*g_deg2rad,  8*g_deg2rad];
	g_instruGripYawCompForceLevel  :ARRAY[1..4] OF INT := [ 20, 40, 70, 101];
	
END_VAR

// ---- GVLs/Instrument/GVL_InstruTypeDefine.TcGVL
// NOTICE：this file would be defined as config file later
{attribute 'global_init_slot' := '49991'}
VAR_GLOBAL CONSTANT
	// only for spatial velocity safety check test
	InstruTypeInfo_TestCartVelInstrument :ST_InstruTypeInfo :=
	(m_InstruID:=1, m_isSingleFinger:=FALSE, m_energyType:=0, m_instruName:='Space Velocity Test Instrument', m_instruNameCH:="空间速度测试器械", m_maxUseNum:=100,
	 m_rodLength:=1.0, m_headLength:=0.0089, m_fingerLength:=0.0195, m_maxGripAngle:=45*g_deg2Rad,
	 m_k1:= 0.859649123, m_k2:=0.947368421, m_k3:=0.775510204,
	 m_rollLimit:=5.5, m_pitchLimit:=80*g_deg2Rad, m_yawLimit:=PI/2, m_normGripTrq := 350,
	 m_instruYawBacklash:=5.5*InstruTypeInfo_TestCartVelInstrument.m_k1*g_deg2Rad, m_instruPitchBachlash:=3*g_deg2Rad);
	 
	InstruTypeInfo_CadiereForceps :ST_InstruTypeInfo :=
	(m_InstruID:=7, m_isSingleFinger:=FALSE, m_energyType:=0, m_instruName:='Cadiere Forceps', m_instruNameCH:="无创抓钳", m_maxUseNum:=10,
	 m_rodLength:=0.5438, m_headLength:=0.0089, m_fingerLength:=0.0195, m_maxGripAngle:=45*g_deg2Rad,
	 m_k1:= 0.859649123, m_k2:=0.947368421, m_k3:=0.775510204,
	 m_rollLimit:=5.5, m_pitchLimit:=80*g_deg2Rad, m_yawLimit:=PI/2, m_normGripTrq := 350,
	 m_instruYawBacklash:=5.5*InstruTypeInfo_CadiereForceps.m_k1*g_deg2Rad, m_instruPitchBachlash:=3*g_deg2Rad);
	 
	InstruTypeInfo_NeedleDriver :ST_InstruTypeInfo :=
	(m_InstruID:=8, m_isSingleFinger:=FALSE, m_energyType:=0, m_instruName:='Large Needle Driver', m_instruNameCH:="持针钳", m_maxUseNum:=10,
	 m_rodLength:=0.5438, m_headLength:=0.0089, m_fingerLength:=0.0096, m_maxGripAngle:=40*g_deg2Rad,
	 m_k1:= 0.824561404, m_k2:=0.947368421, m_k3:=0.808510638,
	 m_rollLimit:=5.5, m_pitchLimit:=80*g_deg2Rad, m_yawLimit:=PI/2, m_normGripTrq := 500,
	 m_instruYawBacklash:=5.5*InstruTypeInfo_NeedleDriver.m_k1*g_deg2Rad, m_instruPitchBachlash:=3*g_deg2Rad);
	 
	InstruTypeInfo_MegaSCNeedleDriver :ST_InstruTypeInfo :=
	(m_InstruID:=9, m_isSingleFinger:=FALSE, m_energyType:=0, m_instruName:='Mega SutureCut Needle Driver', m_instruNameCH:="大号带剪刀持针钳", m_maxUseNum:=10,
	 m_rodLength:=0.5438, m_headLength:=0.01, m_fingerLength:=0.0109, m_maxGripAngle:=40*g_deg2Rad,
	 m_k1:= 1.070175439, m_k2:=0.947368421, m_k3:=0.590163934,
	 m_rollLimit:=5.5, m_pitchLimit:=80*g_deg2Rad, m_yawLimit:=PI/2, m_normGripTrq := 500,
	 m_instruYawBacklash:=5*InstruTypeInfo_MegaSCNeedleDriver.m_k1*g_deg2Rad, m_instruPitchBachlash:=3*g_deg2Rad);
	 
	 InstruTypeInfo_SCNeedleDriver :ST_InstruTypeInfo :=
	(m_InstruID:=10, m_isSingleFinger:=FALSE, m_energyType:=0, m_instruName:='Large SutureCut Needle Driver', m_instruNameCH:="带剪刀持针钳", m_maxUseNum:=10,
	 m_rodLength:=0.5438, m_headLength:=0.01, m_fingerLength:=0.011, m_maxGripAngle:=40*g_deg2Rad,
	 m_k1:= 1.070175439, m_k2:=0.947368421, m_k3:=0.590163934,
	 m_rollLimit:=5.5, m_pitchLimit:=80*g_deg2Rad, m_yawLimit:=PI/2, m_normGripTrq := 500,
	 m_instruYawBacklash:=5*InstruTypeInfo_SCNeedleDriver.m_k1*g_deg2Rad, m_instruPitchBachlash:=3*g_deg2Rad);
	 
	 InstruTypeInfo_RoundTipScissors :ST_InstruTypeInfo :=
	(m_InstruID:=11, m_isSingleFinger:=FALSE, m_energyType:=0, m_instruName:='RoundTip Scissors', m_instruNameCH:="圆头直剪", m_maxUseNum:=10,
	 m_rodLength:=0.5438, m_headLength:=0.0089, m_fingerLength:=0.01102, m_maxGripAngle:=40*g_deg2Rad,
	 m_k1:= 0.842105263, m_k2:=0.947368421, m_k3:=0.791666667,
	 m_rollLimit:=5.5, m_pitchLimit:=80*g_deg2Rad, m_yawLimit:=PI/2, m_normGripTrq := 350,
	 m_instruYawBacklash:=7*InstruTypeInfo_RoundTipScissors.m_k1*g_deg2Rad, m_instruPitchBachlash:=3*g_deg2Rad);
	 
	 InstruTypeInfo_ProGraspForceps :ST_InstruTypeInfo :=
	(m_InstruID:=12, m_isSingleFinger:=FALSE, m_energyType:=0, m_instruName:='Prograsp', m_instruNameCH:="细齿无创抓钳", m_maxUseNum:=10,
	 m_rodLength:=0.5438, m_headLength:=0.01065, m_fingerLength:=0.02773, m_maxGripAngle:=44.5*g_deg2rad,
	 m_k1:= 1.342105263, m_k2:=0.947368421, m_k3:=0.496732026,
	 m_rollLimit:=5.5, m_pitchLimit:=80*g_deg2Rad, m_yawLimit:=PI/2, m_normGripTrq := 350,
	 m_instruYawBacklash:=ASIN((2.8/5.26) * SIN(2.5*InstruTypeInfo_ProGraspForceps.m_k1*g_deg2Rad)), m_instruPitchBachlash:=3*g_deg2Rad);
	 
	 InstruTypeInfo_MarylandForceps :ST_InstruTypeInfo :=
	(m_InstruID:=13, m_isSingleFinger:=FALSE, m_energyType:=2, m_instruName:='Maryland Bipolar Forceps', m_instruNameCH:="双极弧形电凝钳", m_maxUseNum:=10,
	 m_rodLength:=0.5438, m_headLength:=0.01065, m_fingerLength:=0.0195, m_maxGripAngle:=55*g_deg2Rad,
	 m_k1:= 1.070175439, m_k2:=0.947368421, m_k3:=0.590163934,
	 m_rollLimit:=5.5, m_pitchLimit:=80*g_deg2Rad, m_yawLimit:=PI/2, m_normGripTrq := 350,
	 m_instruYawBacklash:=5*InstruTypeInfo_MarylandForceps.m_k1*g_deg2Rad, m_instruPitchBachlash:=3*g_deg2Rad);
	 
	 InstruTypeInfo_FenestratedForceps :ST_InstruTypeInfo :=
	(m_InstruID:=14, m_isSingleFinger:=FALSE, m_energyType:=2, m_instruName:='Fenestrated Bipolar Forceps', m_instruNameCH:="双极鸭嘴电凝钳", m_maxUseNum:=10,
	 m_rodLength:=0.5438, m_headLength:=0.01065, m_fingerLength:=0.0207, m_maxGripAngle:=60.5*g_deg2Rad,
	 m_k1:= 1.070175439, m_k2:=0.947368421, m_k3:=0.590163934,
	 m_rollLimit:=5.5, m_pitchLimit:=80*g_deg2Rad, m_yawLimit:=PI/2, m_normGripTrq := 350,
	 m_instruYawBacklash:=5*InstruTypeInfo_FenestratedForceps.m_k1*g_deg2Rad, m_instruPitchBachlash:=3*g_deg2Rad);
	 
	 InstruTypeInfo_CurvedScissors :ST_InstruTypeInfo :=
	(m_InstruID:=15, m_isSingleFinger:=FALSE, m_energyType:=1, m_instruName:='Monopolar Curved Scissors', m_instruNameCH:="单极弧剪", m_maxUseNum:=10,
	 m_rodLength:=0.5438, m_headLength:=0.0091, m_fingerLength:=0.0130, m_maxGripAngle:=PI/3,
	 m_k1:= 0.842105263, m_k2:=0.947368421, m_k3:=0.75,
	 m_rollLimit:=5.5, m_pitchLimit:=80*g_deg2Rad, m_yawLimit:=PI/2, m_normGripTrq := 350,
	 m_instruYawBacklash:=8*InstruTypeInfo_CurvedScissors.m_k1*g_deg2Rad, m_instruPitchBachlash:=3*g_deg2Rad);
	 
	 InstruTypeInfo_CauteryHook :ST_InstruTypeInfo :=
	(m_InstruID:=16, m_isSingleFinger:=TRUE, m_energyType:=1, m_instruName:='Permanent Cautery Hook', m_instruNameCH:="单极电钩", m_maxUseNum:=10,
	 m_rodLength:=0.5432, m_headLength:=0.00935, m_fingerLength:=0.01668, m_maxGripAngle:=0,
	 m_k1:= 0.964912281, m_k2:= 0.877192982, m_k3:=-0.663636364,
	 m_rollLimit:=5.5, m_pitchLimit:=80*g_deg2Rad, m_yawLimit:=PI/2, m_normGripTrq := 0,
	 m_instruYawBacklash:=7*InstruTypeInfo_CauteryHook.m_k1*g_deg2Rad, m_instruPitchBachlash:=3*g_deg2Rad);
	 
	 InstruTypeInfo_CauterySpatula :ST_InstruTypeInfo :=
	(m_InstruID:=17, m_isSingleFinger:=TRUE, m_energyType:=1, m_instruName:='Permanent Cautery Spatula', m_instruNameCH:="单极电铲", m_maxUseNum:=10,
	 m_rodLength:=0.5432, m_headLength:=0.00935, m_fingerLength:=0.01905, m_maxGripAngle:=0,
	 m_k1:= 0.964912281, m_k2:= 0.877192982, m_k3:=-0.663636364,
	 m_rollLimit:=5.5, m_pitchLimit:=80*g_deg2Rad, m_yawLimit:=PI/2, m_normGripTrq := 0,
	 m_instruYawBacklash:=7*InstruTypeInfo_CauterySpatula.m_k1*g_deg2Rad, m_instruPitchBachlash:=3*g_deg2Rad);
	 
	 InstruTypeInfo_Endoscope :ST_InstruTypeInfo :=
	(m_InstruID:=20, m_isSingleFinger:=FALSE, m_energyType:=0, m_instruName:='Camera', m_instruNameCH:="内窥镜", m_maxUseNum:=100,
	 m_rodLength:=0.49, m_headLength:=0, m_fingerLength:=0, m_maxGripAngle:=0,
	 m_k1:= 1, m_k2:= 1, m_k3:=1,
	 m_rollLimit:=5.5, m_pitchLimit:=1*g_deg2Rad, m_yawLimit:=1*g_deg2Rad, m_normGripTrq := 0,
	 m_instruYawBacklash:=0, m_instruPitchBachlash:=0);
	 
	 InstruTypeInfo_NewEndoscope :ST_InstruTypeInfo :=
	(m_InstruID:=31, m_isSingleFinger:=FALSE, m_energyType:=0, m_instruName:='Camera', m_instruNameCH:="内窥镜", m_maxUseNum:=100,
	 m_rodLength:=0.49, m_headLength:=0, m_fingerLength:=0, m_maxGripAngle:=0,
	 m_k1:= 1, m_k2:= 1, m_k3:=1,
	 m_rollLimit:=5.5, m_pitchLimit:=1*g_deg2Rad, m_yawLimit:=1*g_deg2Rad, m_normGripTrq := 0,
	 m_instruYawBacklash:=0, m_instruPitchBachlash:=0);
	 
	 InstruTypeInfo_UltrasoundKnifeS :ST_InstruTypeInfo :=
	(m_InstruID:=42, m_isSingleFinger:=FALSE, m_energyType:=3, m_instruName:='Ultrasonic Scalpel 45cm', m_instruNameCH:="超声刀 46cm", m_maxUseNum:=1,
	 m_rodLength:=0.46463, m_headLength:=0, m_fingerLength:=0, m_maxGripAngle:=PI/4,
	 m_k1:= 1, m_k2:= 1, m_k3:=1,
	 m_rollLimit:=g_largeNum, m_pitchLimit:=1*g_deg2Rad, m_yawLimit:=1*g_deg2Rad, m_normGripTrq := 350,
	 m_instruYawBacklash:=5*g_deg2Rad, m_instruPitchBachlash:=0);
	 
	 InstruTypeInfo_UltrasoundKnifeU :ST_InstruTypeInfo :=
	(m_InstruID:=43, m_isSingleFinger:=FALSE, m_energyType:=3, m_instruName:='Ultrasonic Scalpel 55cm', m_instruNameCH:="超声刀 55cm", m_maxUseNum:=1,
	 m_rodLength:=0.55225, m_headLength:=0, m_fingerLength:=0, m_maxGripAngle:=PI/4,
	 m_k1:= 1, m_k2:= 1, m_k3:=1,
	 m_rollLimit:=g_largeNum, m_pitchLimit:=1*g_deg2Rad, m_yawLimit:=1*g_deg2Rad, m_normGripTrq := 350,
	 m_instruYawBacklash:=5*g_deg2Rad, m_instruPitchBachlash:=0);
	 
	 InstruTypeInfo_TipUpFenestratedGrasper :ST_InstruTypeInfo :=
	(m_InstruID:=44, m_isSingleFinger:=FALSE, m_energyType:=0, m_instruName:='Tip-Up Fenestrated Grasper', m_instruNameCH:="鸭嘴抓钳", m_maxUseNum:=10,
	 m_rodLength:=0.5438, m_headLength:=0.01065, m_fingerLength:=0.032, m_maxGripAngle:=PI/3,
	 m_k1:= 1.29824561403509, m_k2:=0.947368421052632, m_k3:=0.513513513513513,
	 m_rollLimit:=5.5, m_pitchLimit:=80*g_deg2Rad, m_yawLimit:=PI/2, m_normGripTrq := 350,
	 m_instruYawBacklash:=4*g_deg2Rad, m_instruPitchBachlash:=3*g_deg2Rad);
	 
	 InstruTypeInfo_MegaNeedleDriver :ST_InstruTypeInfo :=
	(m_InstruID:=45, m_isSingleFinger:=FALSE, m_energyType:=0, m_instruName:='Mega Needle Driver', m_instruNameCH:="大号持针钳", m_maxUseNum:=10,
	 m_rodLength:=0.5438, m_headLength:=0.011, m_fingerLength:=0.0130, m_maxGripAngle:=PI/6,
	 m_k1:=1.28070175438596 , m_k2:=0.929824561403509, m_k3:=0.520547945205479,
	 m_rollLimit:=5.5, m_pitchLimit:=80*g_deg2Rad, m_yawLimit:=PI/2, m_normGripTrq := 350,
	 m_instruYawBacklash:=4*g_deg2Rad, m_instruPitchBachlash:=3*g_deg2Rad);
	 
	 InstruTypeInfo_DeBakeyForceps :ST_InstruTypeInfo :=
	(m_InstruID:=46, m_isSingleFinger:=FALSE, m_energyType:=0, m_instruName:='DeBakey Forceps', m_instruNameCH:="微型抓钳", m_maxUseNum:=10,
	 m_rodLength:=0.5438, m_headLength:=0.0089, m_fingerLength:=0.0120, m_maxGripAngle:=PI/6,
	 m_k1:= 0.824561403508772, m_k2:=0.947368421052632, m_k3:=0.808510638297872,
	 m_rollLimit:=5.5, m_pitchLimit:=80*g_deg2Rad, m_yawLimit:=PI/2, m_normGripTrq := 350,
	 m_instruYawBacklash:=4*g_deg2Rad, m_instruPitchBachlash:=3*g_deg2Rad);
	 
	 InstruTypeInfo_BlackDiamondForceps :ST_InstruTypeInfo :=
	(m_InstruID:=47, m_isSingleFinger:=FALSE, m_energyType:=0, m_instruName:='Black Diamond Micro Forceps', m_instruNameCH:="黑钻微型钳", m_maxUseNum:=10,
	 m_rodLength:=0.5438, m_headLength:=0.0089, m_fingerLength:=0.010, m_maxGripAngle:=PI/6,
	 m_k1:= 4.7/5.7, m_k2:=0.947368421052632, m_k3:=0.766,
	 m_rollLimit:=5.5, m_pitchLimit:=80*g_deg2Rad, m_yawLimit:=PI/2, m_normGripTrq := 350,
	 m_instruYawBacklash:=5*g_deg2Rad, m_instruPitchBachlash:=3*g_deg2Rad);
	 
	 InstruTypeInfo_PottsScissors :ST_InstruTypeInfo :=
	(m_InstruID:=48, m_isSingleFinger:=FALSE, m_energyType:=0, m_instruName:='Potts Scissors', m_instruNameCH:="波茨手术剪", m_maxUseNum:=10,
	 m_rodLength:=0.5438, m_headLength:=0.0089, m_fingerLength:=0.0110, m_maxGripAngle:=22*g_deg2Rad,
	 m_k1:= 4.7/5.7, m_k2:=0.947368421052632, m_k3:=0.766,
	 m_rollLimit:=5.5, m_pitchLimit:=80*g_deg2Rad, m_yawLimit:=PI/2, m_normGripTrq := 350,
	 m_instruYawBacklash:=5.5*g_deg2Rad, m_instruPitchBachlash:=3*g_deg2Rad);
	 
	 InstruTypeInfo_CurvedBipolarDissector :ST_InstruTypeInfo :=
	(m_InstruID:=49, m_isSingleFinger:=FALSE, m_energyType:=2, m_instruName:='Curved Bipolar Dissector', m_instruNameCH:="双极分离电凝钳", m_maxUseNum:=10,
	 m_rodLength:=0.5438, m_headLength:=0.01065, m_fingerLength:=0.022, m_maxGripAngle:=PI/4,
	 m_k1:= 1.07017543859649, m_k2:=0.947368421052632, m_k3:=0.59016393442623,
	 m_rollLimit:=5.5, m_pitchLimit:=80*g_deg2Rad, m_yawLimit:=PI/2, m_normGripTrq := 350,
	 m_instruYawBacklash:=4*g_deg2Rad, m_instruPitchBachlash:=3*g_deg2Rad);
	 
	 InstruTypeInfo_MicroBipolarForceps :ST_InstruTypeInfo :=
	(m_InstruID:=50, m_isSingleFinger:=FALSE, m_energyType:=2, m_instruName:='Micro Bipolar Forceps', m_instruNameCH:="双极微型钳", m_maxUseNum:=10,
	 m_rodLength:=0.5438, m_headLength:=0.01065, m_fingerLength:=0.014, m_maxGripAngle:=PI/4,
	 m_k1:= 1.07017543859649, m_k2:=0.947368421052632, m_k3:=0.59016393442623,
	 m_rollLimit:=5.5, m_pitchLimit:=80*g_deg2Rad, m_yawLimit:=PI/2, m_normGripTrq := 350,
	 m_instruYawBacklash:=4*g_deg2Rad, m_instruPitchBachlash:=3*g_deg2Rad);
	 
	 InstruTypeInfo_ForceBipolar :ST_InstruTypeInfo :=
	(m_InstruID:=51, m_isSingleFinger:=FALSE, m_energyType:=5, m_instruName:='Force Bipolar', m_instruNameCH:="强力双极电凝钳", m_maxUseNum:=10,
	 m_rodLength:=0.5438, m_headLength:=0.01065, m_fingerLength:=0.028, m_maxGripAngle:=42*g_deg2Rad,
	 m_k1:= 1.28947368421053, m_k2:=0.947368421052632, m_k3:=0.517006802721088,
	 m_rollLimit:=5.5, m_pitchLimit:=80*g_deg2Rad, m_yawLimit:=PI/2, m_normGripTrq := 220,
	 m_instruYawBacklash:=4*g_deg2Rad, m_instruPitchBachlash:=3*g_deg2Rad);
	 
	 InstruTypeInfo_MicroCauteryHook :ST_InstruTypeInfo :=
	(m_InstruID:=52, m_isSingleFinger:=TRUE, m_energyType:=1, m_instruName:='Micro Permanent Cautery Hook', m_instruNameCH:="小号单极电钩", m_maxUseNum:=10,
	 m_rodLength:=0.5432, m_headLength:=0.00935, m_fingerLength:=0.01668, m_maxGripAngle:=0,
	 m_k1:= 0.964912281, m_k2:= 0.877192982, m_k3:=-0.663636364,
	 m_rollLimit:=5.5, m_pitchLimit:=80*g_deg2Rad, m_yawLimit:=PI/2, m_normGripTrq := 0,
	 m_instruYawBacklash:=8*g_deg2Rad, m_instruPitchBachlash:=3*g_deg2Rad);
	 
	 InstruTypeInfo_CadiereForcepsV2 :ST_InstruTypeInfo :=
	(m_InstruID:=072, m_isSingleFinger:=FALSE, m_energyType:=0, m_instruName:='Cadiere Forceps', m_instruNameCH:="无创抓钳", m_maxUseNum:=19,
	 m_rodLength:=0.5438, m_headLength:=0.0089, m_fingerLength:=0.0195, m_maxGripAngle:=45*g_deg2Rad,
	 m_k1:= 0.859649123, m_k2:=0.947368421, m_k3:=0.775510204,
	 m_rollLimit:=5.5, m_pitchLimit:=80*g_deg2Rad, m_yawLimit:=PI/2, m_normGripTrq := 350,
	 m_instruYawBacklash:=4*g_deg2Rad, m_instruPitchBachlash:=3*g_deg2Rad);
	 
	 InstruTypeInfo_NeedleDriverV2 :ST_InstruTypeInfo :=
	(m_InstruID:=073, m_isSingleFinger:=FALSE, m_energyType:=0, m_instruName:='Large Needle Driver', m_instruNameCH:="持针钳", m_maxUseNum:=16,
	 m_rodLength:=0.5438, m_headLength:=0.0089, m_fingerLength:=0.0096, m_maxGripAngle:=40*g_deg2Rad,
	 m_k1:= 0.824561404, m_k2:=0.947368421, m_k3:=0.808510638,
	 m_rollLimit:=5.5, m_pitchLimit:=80*g_deg2Rad, m_yawLimit:=PI/2, m_normGripTrq := 350,
	 m_instruYawBacklash:=4*g_deg2Rad, m_instruPitchBachlash:=3*g_deg2Rad);
	 
	 InstruTypeInfo_MarylandForcepsV2 :ST_InstruTypeInfo :=
	(m_InstruID:=074, m_isSingleFinger:=FALSE, m_energyType:=2, m_instruName:='Maryland Bipolar Forceps', m_instruNameCH:="双极弧形电凝钳", m_maxUseNum:=15,
	 m_rodLength:=0.5438, m_headLength:=0.01065, m_fingerLength:=0.0195, m_maxGripAngle:=55*g_deg2Rad,
	 m_k1:= 1.070175439, m_k2:=0.947368421, m_k3:=0.590163934,
	 m_rollLimit:=5.5, m_pitchLimit:=80*g_deg2Rad, m_yawLimit:=PI/2, m_normGripTrq := 350,
	 m_instruYawBacklash:=4*g_deg2Rad, m_instruPitchBachlash:=3*g_deg2Rad);
	  
	 InstruTypeInfo_FenestratedForcepsV2 :ST_InstruTypeInfo :=
	(m_InstruID:=075, m_isSingleFinger:=FALSE, m_energyType:=2, m_instruName:='Fenestrated Bipolar Forceps', m_instruNameCH:="双极鸭嘴电凝钳", m_maxUseNum:=15,
	 m_rodLength:=0.5438, m_headLength:=0.01065, m_fingerLength:=0.0207, m_maxGripAngle:=55*g_deg2Rad,
	 m_k1:= 1.070175439, m_k2:=0.947368421, m_k3:=0.590163934,
	 m_rollLimit:=5.5, m_pitchLimit:=80*g_deg2Rad, m_yawLimit:=PI/2, m_normGripTrq := 350,
	 m_instruYawBacklash:=4*g_deg2Rad, m_instruPitchBachlash:=3*g_deg2Rad);
	 
	 g_instruTypeNum :INT :=25;
	 g_instruTypePool :ARRAY[1..g_instruTypeNum] OF ST_InstruTypeInfo :=
	 [InstruTypeInfo_TestCartVelInstrument, InstruTypeInfo_CadiereForceps, 	InstruTypeInfo_NeedleDriver,  		InstruTypeInfo_MegaSCNeedleDriver, 	InstruTypeInfo_SCNeedleDriver,
	  InstruTypeInfo_RoundTipScissors,	InstruTypeInfo_ProGraspForceps,		InstruTypeInfo_MarylandForceps,		InstruTypeInfo_FenestratedForceps,
	  InstruTypeInfo_CurvedScissors,	InstruTypeInfo_CauteryHook,	 		InstruTypeInfo_CauterySpatula, 		InstruTypeInfo_Endoscope, InstruTypeInfo_NewEndoscope,
	  InstruTypeInfo_UltrasoundKnifeU, 	InstruTypeInfo_UltrasoundKnifeS,	InstruTypeInfo_TipUpFenestratedGrasper, 		InstruTypeInfo_MegaNeedleDriver, 
	  InstruTypeInfo_DeBakeyForceps, 	InstruTypeInfo_BlackDiamondForceps, 	InstruTypeInfo_PottsScissors, 	InstruTypeInfo_CurvedBipolarDissector,
	  InstruTypeInfo_MicroBipolarForceps,InstruTypeInfo_ForceBipolar, InstruTypeInfo_MicroCauteryHook];
	  
	 // map derivated instrument to normal type, which is different with normal instument only with ID 
	 g_derivedInstruNum :INT := 33;
	 g_InstruTypeMap:ARRAY[1..g_derivedInstruNum] OF Vec3i :=
	 [[307, 7, 0], [308, 8, 0], [309, 9, 0], [310, 10, 0], [311, 11, 0], [312, 12, 0], [313, 13, 0], [314, 14, 0], 
	  [315, 15, 0], [316, 16, 0], [317, 17, 0], [320, 31, 0], [321, 31, 0],
	  [72, 7, 19], [73, 8, 16], [74, 13, 15], [75, 14, 15],
	  [91, 7, 30], [92, 8, 30], [93, 9, 30],[94, 10, 30], [95, 12, 30], [96, 13, 30],[97, 14, 30], [98, 15, 30], [99, 16, 30],[100, 17, 30], [101, 44, 30], [102, 45, 30],[103, 49, 30], [104, 50, 30],
	  [166, 31, 0],[167, 31, 0]];
END_VAR

// ---- GVLs/SlaveArms/GVL_SlaveArmDynamics.TcGVL
{attribute 'global_init_slot' := '49992'}
{attribute 'qualified_only'}
// Robot5 --dynamic parameters of slave arms
VAR_GLOBAL CONSTANT
	
	// arm gravity parameters
(*graParam=[ 9.8*m5,...
           0.41601*m2 + 0.41601*m3 + 0.0000216012*m4 + 0.0000216012*m5 + 9.8*mx1 - 1.3639*mx3 - 9.70463*my3,...
           9.8*mz2 - 9.8*my5 - 9.8*my1 + 9.8*mz3 + 9.8*mz4,...
           2.19651*m3 + 2.19651*m4 + 0.00000258969*m5 + 8.64766*mx2 - 4.61063*my2 + 9.8*my4 + 9.8*mz5,...
          1.1711*m3 + 1.1711*m4 + 0.00000122416*m5 + 4.61063*mx2 - 9.8*mx4 - 9.8*mx5 + 8.64766*my2]'
*)			
	// robot No.4
	g_gravityParam :ARRAY[1..g_sArmNum,1..5] OF REAL := [5(0)];
	 
	g_gravityTrocar :ARRAY[1..5] OF REAL :=[0.1661, -0.4124,  0.0964,   -0.7987,   -0.6999 ];
	g_gravityInstrument :ARRAY[1..5] OF REAL :=[ 3.1217,  -0.3099,   0.0778,   -1.2498,   -0.8041];
	g_gravityEndoscope :ARRAY[1..5] OF REAL :=[10.8619,  -0.8575,   -1.0274,   -0.2425,   -0.0869];
	
	// joint friction(with instrument mounted)
	g_slaveJntFriction :ARRAY[1..g_sArmNum, 1..g_sJntNum] OF LREAL :=
			[ 0,    0,    0,  0.03, 0.03, 0.03, 0.03, 0];
			  
	//################ DO NOT modify parameters below ###########################
	//################ dynamic reference model parameters below ###########################
	// link mass [m1, m2, m3, m4, m5]
	g_linkMass :ARRAY[1..5] OF LREAL :=[5.6565, 1.4613, 1.149, 1.5362, 0.6679] ;
	
	// lin center of amss
	g_linkCOM :ARRAY[1..5,1..3] OF LREAL :=  [ 0.0566,    0.0302,   -0.4685,
											   0.1191,   -0.0011,   -0.0588,
											   0.1238,    0.0003,   -0.0120,
											   0.0427,    0.0924,   -0.0004,
											   -0.0262,        0,   -0.0292];
	// link  inertial
    // [Ixx,Iyy,Izz, Ixy,Ixz, Iyz]
 	g_linkInertia :ARRAY[1..5,1..6] OF LREAL :=[0.0735,    0.0738,    0.0144,    0.0016,   -0.0000,   -0.0079,
												0.0016,    0.0190,    0.0185,         0,    0.0027,         0,
											   0.0009,    0.0167,    0.0166,         0,    0.0012,         0,
												0.0009,    0.0167,    0.0166,         0,    0.0012,         0,
											  0.0009,    0.0167,    0.0166,         0,    0.0012,         0];

	
	//  motor inertial at link size
	g_motorInertia :ARRAY[1..3] OF LREAL := [0.00004487, 0.00004487, 0.0000002280];
	
END_VAR

// ---- GVLs/SlaveArms/GVL_SlaveControlParameters.TcGVL
{attribute 'global_init_slot' := '49991'}
VAR_GLOBAL CONSTANT
	// slave arm joint position controller parameters
	//g_posKp :ARRAY[1..g_sJntNum] OF LREAL :=[2000.0, 2000.0, 18000.0, 5(5)];
	//g_posKd :ARRAY[1..g_sJntNum] OF LREAL :=[200.0, 200.0, 1800.0, 5(0.25)];
	//g_posKi :ARRAY[1..g_sJntNum] OF LREAL :=[20000.0, 20000.0, 30000.0, 5(10.0)];
	//g_posKiLimit :ARRAY[1..g_sJntNum] OF LREAL :=[2500,2500,  250, 5(75)];// define in current
	//g_posCtrlLimit :ARRAY[1..g_sJntNum] OF LREAL :=[5600,5600,  500, 5(200)];// define in current
	g_posKp :ARRAY[1..g_sJntNum] OF LREAL :=[2000.0, 2000.0, 5000.0, 5(2)];
	g_posKd :ARRAY[1..g_sJntNum] OF LREAL :=[200.0, 200.0, 300.0, 5(0.02)];
	g_posKi :ARRAY[1..g_sJntNum] OF LREAL :=[20000.0, 20000.0, 20000.0, 5(5.0)];
	g_posKiLimit :ARRAY[1..g_sJntNum] OF LREAL :=[2500,2500,  500, 5(400)];// define in current
	g_posCtrlLimit :ARRAY[1..g_sJntNum] OF LREAL :=[5600,5600,  1300, 5(500)];// define in current
	
	// control tolerance
	g_jntCtrlAngTolLow :LREAL :=0.2*g_deg2Rad;
	g_jntCtrlAngTolHigh :LREAL :=2*g_deg2Rad;
	g_cartCtrlPosTolLow :LREAL :=0.0002;
	g_cartCtrlOriTolLow :LREAL :=0.2*g_deg2Rad;
	g_cartCtrlPosTolHigh :LREAL :=0.001;
	g_cartCtrlOriTolHigh :LREAL :=2*g_deg2Rad;
	
	// filter cut-off frequency for velocity and torque
	g_curJntVelLpfCutoffFreq :LREAL := 30;
	g_cmdJntTrqLpfCutoffFreq :LREAL := 300;
	g_curJntTrqLpfCutoffFreq :LREAL := 300;
		
	// controller would keep command unchanged when error 
	// between command and current value is less than this value
	g_jntCtrlErrForCmdHold :LREAL :=1.0*g_deg2Rad;
	
	// joint is assumed to be static if velocity is less than this value
	g_jntStaticVelThres :LREAL :=0.2*g_deg2Rad;
	
	// joint velocity threshold for full friction compensation
	g_fullFrictionVel :LREAL :=2.0*g_deg2Rad;
	
	// friciton compensation scael
	g_frictionCompScale :LREAL := 0.8;
	
END_VAR

// ---- GVLs/SlaveArms/GVL_SlaveJointEncoderCaliData.TcGVL
{attribute 'qualified_only'}
// Robot5 --joints parameters of slave arms
VAR_GLOBAL CONSTANT
	// absolute encoder value at minimal joint positon
	g_minLinkEncoder :ARRAY[1..g_sArmNum, 1..g_sJntNum] OF DINT :=
		[0, 0, 0, 0, 0, 0, 0, 0];
		 
	// absolute encoder value at maximum joint positon
	g_maxLinkEncoder :ARRAY[1..g_sArmNum, 1..g_sJntNum] OF DINT :=
		[0, 0, 0, 0, 0, 0, 0, 0];
END_VAR
VAR_GLOBAL RETAIN
	
	// absolute encoder value at calibrated positon
	g_caliLinkEncoder :ARRAY[1..g_sArmNum, 1..g_sJntNum] OF DINT :=
		[0, 0, 0,33629,53410,37426,768,20369];
END_VAR
VAR_GLOBAL CONSTANT
	
	 // if absolute encoder value cross zeros within joint motion range
	 // NOTICE: joint 7 is always 0.
	g_linkEncZeroCross :ARRAY[1..g_sArmNum, 1..g_sJntNum] OF INT :=
		[1, 0, 1, 1, 1, 1, 1, 1];
		 
	 // joint SDO address
	g_slaveArmNetID: ARRAY[1..g_sArmNum] OF T_AmsNetId:=['192.168.2.195.4.1'];//['192.168.3.122.5.1'];
	g_slaveJointNetPort:ARRAY[1..g_sArmNum,1..g_sJntNum] OF UINT :=[
		1006,	1007,	1008,	2(1001),	3(1002)];
	g_slaveLEDNetPort:ARRAY[1..g_sArmNum] OF UINT :=[1001];
		
//################ DO NOT modify parameters below ###########################
	// abolute encoder expanded limit buffer in case there is calibrtion error at limit position
	g_linkEncLimitBuffer : DINT := 100000;
	
	// absolute encoder direction
	g_asbEncoderDir :ARRAY[1..g_sJntNum] OF INT :=[1, -1, 1, -1, -1, -1, -1, -1];
	
	// flag if joint can rotate multiple cycles
	g_multipleCyclesJoint :ARRAY[1..g_sArmNum, 1..g_sJntNum] OF INT :=
		[0, 0, 0, 1, 1, 1, 1, 1];
		 
	// joint position at link encoder calibrated point
	g_linkEncCaliJntPos :ARRAY[1..g_sJntNum] OF LREAL :=
		[0.0, -PI/2, 0.581633, 5(-PI/2)];

	
END_VAR

// ---- GVLs/SlaveArms/GVL_SlaveMotorParameters.TcGVL
{attribute 'global_init_slot' := '49991'}
{attribute 'qualified_only'}
VAR_GLOBAL CONSTANT
	// encoder resolution
	g_incEncoderRes :ARRAY[1..g_sJntNum] OF DINT :=[2(65536),4096,5(2048)];
	g_absEncoderRes :ARRAY[1..g_sJntNum] OF DINT :=[2(131072),6(65536)];
	
	// reduction ratio
	g_motorReduction :ARRAY[1..g_sJntNum] OF LREAL :=[ 81,81,  2*PI/0.006,5(221.0/11)];//(66.0/10)*2*pi/0.010,5(388125.0/4693)];
	g_absEncoderReduction :ARRAY[1..g_sJntNum] OF LREAL :=[2(1.0), 2*PI/0.64, 5(1.0)];
	
	// motor parameters
	g_motorTrqConst :ARRAY[1..g_sJntNum] OF LREAL :=[0.9/5.6,0.9/5.6, 0.032,5(0.0303)];

	// motor encoder direction
	g_motorDir :ARRAY[1..g_sJntNum] OF INT :=[-1, 1, -1, 1, 1, 1, 1, 1];
																 
	// joint position limit
	g_minJntPos: ARRAY[1..g_sJntNum] OF LREAL:=[-2.7,	-1.5-pi/2,	0.23, 	5(-g_largeNum)];	
	g_maxJntPos: ARRAY[1..g_sJntNum] OF LREAL:=[2.7,	1.13-pi/2, 	0.58, 		5(g_largeNum)];
	
	// DH joint position limit
	//NOTE: wrist pitch and yaw angle is reset after instrument is mounted 
	g_minDHJntPos : ARRAY[1..6] OF LREAL :=[-2.7,	-1.5-pi/2,	0.235, -5.5, -PI/2 - 75*g_deg2Rad , -PI/2];
	g_maxDHJntPos : ARRAY[1..6] OF LREAL :=[2.7,	1.13-pi/2, 	0.575, 5.5, -PI/2 + 75*g_deg2Rad, PI/2];
	
	// joint velocity limit
	g_maxJntVel :ARRAY[1..g_sJntNum] OF LREAL :=[1.3, 1.3, 0.5, 5(4*pi)];
	g_motorPID:ARRAY[1..g_sJntNum,1..6] OF INT:=[18(0),
												 10000,8000,400,20,100,540,
												 10000,8000,400,20,100,540,
												 10000,8000,400,20,100,540,
												 10000,8000,400,20,100,540,
												 10000,8000,400,20,100,540];	
END_VAR

VAR_GLOBAL
	g_motorMaxCurrent :ARRAY[1..g_sJntNum] OF LREAL :=[ 5600,5600,  1300, 5(800)];//mA
END_VAR

// ---- FBs_Robots/FB_Instrument.TcPOU
FUNCTION_BLOCK FB_Instrument



VAR
	// instrument type
	m_instruType : 	E_InstrumentType := InstruType_UNKNOWM;
	
	// instrument type info
	m_instruTypeInfo : 	ST_InstruTypeInfo;
	
	//The state and parameters readed from the instrument
	m_onChipData:ST_InstruOnChipData;
	
	// current and max allowed read tries
	m_curReadTries :INT :=0;
	m_maxReadTries :INT := 20;
	
	//IP of operating arm
	m_armNetId:T_AmsNetId; 	
	
	//Joint port number
	m_jointInstruAddr:UINT;	
	
	//LED port address
	m_LEDAddr:UINT;		

	// joint position when instrument is at ZERO posture
	m_jntPosOffset:Vec8d;
	
	// instrument wrist DH joint limit
	m_wristMinDHJntPos :Vec3d;
	m_wristMaxDHJntPos :Vec3d;
	
	// reduction from motor joint to endoscope rotate joint
	m_endoscopeRotateReduction :LREAL := 2.0/3.0;
	
	//endoscope type
	m_curEndoscopeType :E_EndoscopeType:=EndoScopeType_30;
	m_nextEndoscopeType :E_EndoscopeType:=EndoScopeType_30;
	
	//endoscope posutre
	m_curEndoscopePosture :E_EndoscopePosture:=EndoscopePosture_HeadDown;
	m_nextEndoscopePosture :E_EndoscopePosture:=EndoscopePosture_HeadDown;
	
	// udint code for zero position
	m_zeroPosCode : UDINT;
	
	// joint4 zero position, which is supposed to be a contant value
	m_jnt4ZeroPos :LREAL := 5.7;
	
	//reset arm  LED flag
	m_resetArmLEDFlag : BOOL :=TRUE;
	
	// variables used to read instrument information
	m_Step:INT;
	m_Value:UDINT;
	m_ReadDelay:TON;
	m_DealyTime:TIME:=T#0.5S;
	m_IDReadResult:UDINT;
	m_IDResult:ULINT;
	m_SeriesReadResult:UDINT;
	m_PosReadResult:UDINT;
	m_PosL1,m_PosL2,m_PosL3:UDINT;
	m_signL1,m_signL2,m_signL3:UDINT;
	m_UsageReadResult:ULINT;
	m_InstruUsageToLED:ULINT;
	m_purposeReadResult:ULINT;
	m_HaveRecord:BOOL;
	m_SdoWrite:FB_EcCoESdoWrite;
	m_SdoRead:FB_EcCoESdoRead;
	
	//variables used to read-write instrument number of use
	m_useNumStep : INT;
	m_ReadNumDelay:TON;
	m_useNumReadResult:ULINT;
	m_useNumSendToLED:ULINT;
	
	// rising edge generator for instrument information reading
	m_writeLDP:R_TRIG;
	m_SDOStep: INT;
	m_fbTon_Step: ARRAY[0..5] OF TON;
	value: ULINT;
	m_purposeMode:UINT;
	m_StepRFID:INT;
	m_ReadDelayRFID:TON;
	
	// max Usage Counts of derived intruments
	m_mapInstruMaxUsage :INT :=0;
END_VAR

METHOD PUBLIC addNumOfUseToChip : BOOL
VAR
END_VAR
value:=16#40000000;
addNumOfUseToChip:=FALSE;
m_SdoWrite(sNetId:= m_ArmNetId, nSlaveAddr:= m_JointInstruAddr, nSubIndex:= 0, nIndex:= 16#6094, pSrcBuf:= ADR(value), cbBufLen:= SIZEOF(value), bExecute:= TRUE, );
IF NOT m_SdoWrite.bBusy THEN
	m_SdoWrite(bExecute:=FALSE);
	addNumOfUseToChip:=TRUE;
END_IF
END_METHOD

METHOD PROTECTED checkInstruType : BOOL
VAR_INPUT
END_VAR
VAR
	i:INT;
END_VAR
// search instrument type
checkInstruType :=FALSE;
 //m_onChipData.m_InstruID := InstruType_UltrasoundKnifeS;
FOR i:=1 TO g_instruTypeNum DO 
	IF g_instruTypePool[i].m_InstruID = m_onChipData.m_InstruID THEN
		checkInstruType:=TRUE;
		m_instruTypeInfo := g_instruTypePool[i];
		IF m_mapInstruMaxUsage>0 THEN 
			m_instruTypeInfo.m_maxUseNum:=m_mapInstruMaxUsage;
		END_IF
		EXIT;
	END_IF
END_FOR

// return directly if instrument ID is invalid
IF NOT(checkInstruType) THEN
	RETURN;
END_IF
m_instruType := m_onChipData.m_InstruID;

// update DH joint limit
m_wristMinDHJntPos[1]:=-m_instruTypeInfo.m_rollLimit;
m_wristMaxDHJntPos[1]:=m_instruTypeInfo.m_rollLimit;
m_wristMinDHJntPos[2]:=-m_instruTypeInfo.m_pitchLimit-pi/2;
m_wristMaxDHJntPos[2]:=m_instruTypeInfo.m_pitchLimit-pi/2;
m_wristMinDHJntPos[3]:=-m_instruTypeInfo.m_yawLimit;
m_wristMaxDHJntPos[3]:=m_instruTypeInfo.m_yawLimit;
END_METHOD

METHOD PUBLIC clearNumOfUseToChip : BOOL
VAR
END_VAR
value:=16#80000000;
clearNumOfUseToChip:=FALSE;
m_SdoWrite(sNetId:= m_ArmNetId, nSlaveAddr:= m_JointInstruAddr, nSubIndex:= 0, nIndex:= 16#6094, pSrcBuf:= ADR(value), cbBufLen:= SIZEOF(value), bExecute:= TRUE, );
IF NOT m_SdoWrite.bBusy THEN
	m_SdoWrite(bExecute:=FALSE);
	clearNumOfUseToChip:=TRUE;
END_IF
END_METHOD

PROPERTY curScopePosture : E_EndoscopePosture
GET
curScopePosture:= m_curEndoscopePosture;
END_GET
SET
m_curEndoscopePosture := curScopePosture;
END_SET
END_PROPERTY

PROPERTY curScopeType : E_EndoscopeType
GET
curScopeType := m_curEndoscopeType;
END_GET
SET
m_curEndoscopeType := curScopeType;
END_SET
END_PROPERTY

METHOD PUBLIC gripAngleMap : BOOL
VAR_INPUT
	// master gripper angle
	i_masterGripAng :LREAL;
END_VAR

VAR_OUTPUT
	// slave instrument gripper angle
	o_instruGripAngle :LREAL;
	
	// slave instrument grip force	
	o_instruGripForceLevel :LREAL;
END_VAR

VAR
	gripLevel :REAL;
END_VAR
// suppose finger is  closed and zero force if instrument has only one finger
IF m_instruTypeInfo.m_isSingleFinger THEN
	o_instruGripAngle := 0;
	o_instruGripForceLevel:= 0;
	RETURN;
END_IF 

// finger closed and force applied
IF i_masterGripAng < g_masterGripForceStartAng THEN
	o_instruGripAngle := g_minSlaveGripAngle;
	// NOTE: force is applied from 50%，as minimum gripper angle already apply some sort of force
	o_instruGripForceLevel := 50+50*(g_masterGripForceStartAng - i_masterGripAng)/(g_masterGripForceStartAng - g_minMasterGripAngle);
// finger open
ELSE
	o_instruGripAngle := (g_maxMasterGripAngle - i_masterGripAng)/(g_maxMasterGripAngle - g_masterGripForceStartAng);
	o_instruGripAngle :=m_instruTypeInfo.m_maxGripAngle - o_instruGripAngle * (m_instruTypeInfo.m_maxGripAngle - g_minSlaveGripAngle);
	o_instruGripAngle := LIMIT(g_minSlaveGripAngle, o_instruGripAngle, m_instruTypeInfo.m_maxGripAngle );
	o_instruGripForceLevel:=0;
END_IF
END_METHOD

METHOD PUBLIC init : BOOL
VAR_INPUT
	armIdx :INT;
END_VAR
VAR
	i:INT;
END_VAR
//Update the IP and port number of the operating arm
m_armNetId:=GVL_SlaveJointEncoderCaliData.g_slaveArmNetID[armIdx];
m_jointInstruAddr:=GVL_SlaveJointEncoderCaliData.g_slaveJointNetPort[armIdx,4];
m_LEDAddr := GVL_SlaveJointEncoderCaliData.g_slaveLEDNetPort[armIdx];

// init joint motion range
FOR i:=1 TO 3 DO
	m_wristMinDHJntPos[i]:=GVL_SlaveMotorParameters.g_minDHJntPos[i+3];
	m_wristMaxDHJntPos[i]:=GVL_SlaveMotorParameters.g_maxDHJntPos[i+3];
END_FOR
END_METHOD

METHOD PUBLIC initInstruJntPos : BOOL
VAR_INPUT
	m_curJntPos :Vec8d;
END_VAR

VAR
	i:INT;
END_VAR
FOR i := 4 TO 8 BY 1 DO
	m_jntPosOffset[i]:=m_curJntPos[i];
END_FOR
END_METHOD

// convert motor joint position to DH joint position
METHOD PUBLIC instruFK : BOOL
VAR_IN_OUT CONSTANT
	// motor joint position of slave arm
	i_jntPos :Vec8d;
END_VAR

VAR_IN_OUT
	// instrument DH  joint positon
	r_DHJntPos :Vec6d;

	// gripper angle
	r_gripAngle :LREAL;
END_VAR

VAR
	jntPosL1,jntPosL2,jntPosL3,jntPosL4,jntPosL5 :LREAL;
	gripAngle:LREAL;
	kx,ky,kz, k13, k23,openAngleDir:LREAL;
END_VAR
r_DHJntPos[1]:=i_jntPos[1];
r_DHJntPos[2]:=i_jntPos[2];
r_DHJntPos[3]:=i_jntPos[3];

// kinematic variables
openAngleDir:=-1;
kx:=-1;
ky:=m_instruTypeInfo.m_k2;
kz:=m_instruTypeInfo.m_k1;
k13:=m_instruTypeInfo.m_k3;
k23:=m_instruTypeInfo.m_k3;


// ################## endoscope ############################
IF m_instruType = InstruType_endoscope THEN
	r_DHJntPos[4]:=m_endoscopeRotateReduction*(i_jntPos[8]-m_jntPosOffset[8]);
	IF m_curEndoscopeType = EndoScopeType_30 THEN
		r_DHJntPos[5]:=-pi/2+30*g_deg2Rad;
	ELSE
		r_DHJntPos[5]:=-pi/2;
	END_IF
	r_DHJntPos[6]:=0;
	RETURN;
END_IF

// ################## ultrosonic knief ############################
IF m_instruType = InstruType_UltrasoundKnifeS OR m_instruType = InstruType_UltrasoundKnifeU THEN
	r_DHJntPos[4]:=-(i_jntPos[8]-m_jntPosOffset[8])/kx;
	r_DHJntPos[5]:=-pi/2;
	r_DHJntPos[6]:=0;
	r_gripAngle:=ultrasoundKnifeGripAngleFK(i_jntPos[6]-m_jntPosOffset[6]);
	RETURN;
END_IF


//#################### instrument forward kinematic ############
// convert motor joint position to instrument joint position
jntPosL1:=(i_jntPos[4]-m_jntPosOffset[4]);
jntPosL2:=(i_jntPos[5]-m_jntPosOffset[5]);
jntPosL3:=(i_jntPos[6]-m_jntPosOffset[6]);
jntPosL4:=-(i_jntPos[7]-m_jntPosOffset[7]);
jntPosL5:=-(i_jntPos[8]-m_jntPosOffset[8]);

// diable L1 if instrument is single finger
IF m_instruTypeInfo.m_isSingleFinger THEN
	jntPosL1 := -jntPosL2;
END_IF

// instrument FK in local coordinate
r_DHJntPos[4]:=jntPosL4/kx;
r_DHJntPos[5]:=jntPosL3/ky;
r_DHJntPos[6]:=(jntPosL1-jntPosL2-2*r_DHJntPos[5]*k13*kz)/(2*openAngleDir*kz);

// convert instrument rotation to arm DH joint position
r_DHJntPos[5]:=-r_DHJntPos[5]-pi/2;
r_DHJntPos[6]:=-r_DHJntPos[6];

// grip angle
gripAngle:=(jntPosL1+jntPosL2)/(openAngleDir*kz);

//################### gripper angle handle #################
IF (InstruType_ProGraspForceps=m_instruType OR InstruType_ForceBipolar=m_instruType) THEN//细齿无创抓钳
	proGrsapForcepsGripAngleFK(frontAngle:= gripAngle, endAngle=> r_gripAngle);

ELSIF (InstruType_CauteryHook = m_instruType OR InstruType_CauterySpatula = m_instruType) THEN//单级电钩
	r_gripAngle:=0;
ELSE
	r_gripAngle:=gripAngle;
END_IF
END_METHOD

METHOD InstruIDMap : INT
VAR
	i:INT;
END_VAR
m_mapInstruMaxUsage:=0;
FOR i:=1 TO g_derivedInstruNum DO
	IF g_InstruTypeMap[i][1] =  m_onChipData.m_InstruID THEN 
		m_onChipData.m_InstruID := g_InstruTypeMap[i][2];
		m_mapInstruMaxUsage:=g_InstruTypeMap[i][3];
	END_IF
END_FOR
END_METHOD

METHOD PROTECTED InstruIDRecord :ARRAY [1..100] OF  ULINT
VAR_INPUT
	i_NewValue:ULINT;
	i_ArrayData:ARRAY [1..100] OF ULINT;
END_VAR

VAR
	k1:INT;
	Have_Data:BOOL;
END_VAR
FOR k1:= 1 TO 100 BY 1 DO
	IF i_NewValue=i_ArrayData[k1] THEN
		Have_Data:=TRUE;
		EXIT;
	ELSE
		Have_Data:=FALSE;
	END_IF
END_FOR

IF Have_Data=FALSE THEN
	FOR k1:= 1 TO 99 BY 1 DO
		InstruIDRecord[k1+1]:=i_ArrayData[k1];
	END_FOR
	InstruIDRecord[1]:=i_NewValue;
ELSE
	InstruIDRecord:=i_ArrayData ;
END_IF
END_METHOD

METHOD PUBLIC instruIK : BOOL
VAR_INPUT
	// DH  joint positon
	i_DHJntPos :Vec6d;

	// gripper angle
	i_gripAngle :LREAL;
	
END_VAR
VAR_OUTPUT
	o_jntPos:Vec8d;
END_VAR
VAR
	gripAngle:LREAL;
	i:INT;
	rot_x:lreal;
	rot_y:lreal;
	rot_z:lreal;

	kx,ky,kz,k13,k23:LREAL;
	d,ra:LREAL;
	
	m_gripAnglePbox:Vec8d;

END_VAR
o_jntPos[1] := i_DHJntPos[1];
o_jntPos[2] := i_DHJntPos[2];
o_jntPos[3] := i_DHJntPos[3];

// kinematic variables
d:=-1;
kx:=-1;
ky:=m_instruTypeInfo.m_k2;
kz:=m_instruTypeInfo.m_k1;
k13:=m_instruTypeInfo.m_k3;
k23:=m_instruTypeInfo.m_k3;

// ################## endoscope ############################
IF m_instruType = InstruType_endoscope THEN
	o_jntPos[8] := i_DHJntPos[4]/m_endoscopeRotateReduction + m_jntPosOffset[8];
	o_jntPos[4]:=0;
	o_jntPos[5]:=0;
	o_jntPos[6]:=0;
	o_jntPos[7]:=0;
	RETURN;
END_IF

//################### gripper angle handle #################
IF (InstruType_ProGraspForceps=m_instruType OR InstruType_ForceBipolar=m_instruType) THEN//细齿无创抓钳
	proGrsapForcepsGripAngleIK(endAngle:= i_gripAngle, frontAngle=> gripAngle);
	
ELSIF (InstruType_CauteryHook = m_instruType OR InstruType_CauterySpatula = m_instruType)  THEN//单级电钩\电铲
	gripAngle:=0;
	
ELSE
	gripAngle:=i_gripAngle;
END_IF

// ################# instrument inverse kinematic ##############
// convert arm DH joint position to  instrument rotation
rot_x:=i_DHJntPos[4];
rot_y:=-i_DHJntPos[5]-pi/2;
rot_z:=-i_DHJntPos[6];

// ################## ultrosonic knief ############################
IF InstruType_UltrasoundKnifeS = onChipData.m_InstruID OR InstruType_UltrasoundKnifeU = onChipData.m_InstruID THEN
	m_gripAnglePbox[4]:=0;
	m_gripAnglePbox[5]:=0;
	m_gripAnglePbox[6]:=ultrasoundKnifeGripAngleIK(gripAngle); 
	m_gripAnglePbox[7]:=rot_x*kx;
	m_gripAnglePbox[8]:=rot_x*kx;
ELSE
	m_gripAnglePbox[7]:=rot_x*kx;
	m_gripAnglePbox[6]:=rot_y*ky;
	ra:=gripAngle;
	m_gripAnglePbox[4]:=rot_y*k13*kz+d*rot_z*kz+d*ra*kz/2;
	m_gripAnglePbox[5]:=-rot_y*k23*kz-d*rot_z*kz+d*ra*kz/2;
END_IF

// convert instrument joint position to motor joint position
o_jntPos[4] := m_gripAnglePbox[4] + m_jntPosOffset[4];
o_jntPos[5] := m_gripAnglePbox[5] + m_jntPosOffset[5];
o_jntPos[6] := m_gripAnglePbox[6] + m_jntPosOffset[6];
o_jntPos[7] := -m_gripAnglePbox[7] + m_jntPosOffset[7];
o_jntPos[8] := -m_gripAnglePbox[8] + m_jntPosOffset[8];
END_METHOD

// convert motor joint velocity to DH joint velocity
METHOD PUBLIC instruJntVelFK : BOOL
VAR_IN_OUT CONSTANT
	// motor joint velocity of slave arm
	i_jntVel :Vec8d;
END_VAR

VAR_IN_OUT
	// instrument DH  joint velocity
	r_DHJntVel :Vec6d;
END_VAR

VAR
	kx,ky,kz, k13, k23,openAngleDir:LREAL;
END_VAR
r_DHJntVel[1]:=i_jntVel[1];
r_DHJntVel[2]:=i_jntVel[2];
r_DHJntVel[3]:=i_jntVel[3];

// kinematic variables
openAngleDir:=-1;
kx:=-1;
ky:=m_instruTypeInfo.m_k2;
kz:=m_instruTypeInfo.m_k1;
k13:=m_instruTypeInfo.m_k3;
k23:=m_instruTypeInfo.m_k3;

r_DHJntVel[4]:=-i_jntVel[7]/kx;
r_DHJntVel[5]:=i_jntVel[6]/ky;
r_DHJntVel[6]:=(i_jntVel[4]-i_jntVel[5]-2*r_DHJntVel[5]*k13*kz)/(2*openAngleDir*kz);
r_DHJntVel[5]:=-r_DHJntVel[5];
r_DHJntVel[6]:=-r_DHJntVel[6];
END_METHOD

METHOD PROTECTED InstruSreiesFind : BOOL
VAR_INPUT
	i_NewValue:ULINT;
	i_ArrayData:ARRAY [1..100] OF ULINT;
	
END_VAR

VAR
	k1:INT;
END_VAR
InstruSreiesFind:=FALSE;
FOR k1:= 1 TO 100 BY 1 DO
	IF i_NewValue=i_ArrayData[k1] THEN
		InstruSreiesFind:=TRUE;
		EXIT;
	ELSE
		InstruSreiesFind:=FALSE;
	END_IF
END_FOR
END_METHOD

PROPERTY PUBLIC instruType : E_InstrumentType
GET
instruType := m_instruType;
END_GET
END_PROPERTY

PROPERTY instruTypeInfo :REFERENCE TO ST_InstruTypeInfo
GET
instruTypeInfo ref=m_instruTypeInfo;
END_GET
END_PROPERTY

PROPERTY nextScopePosture : E_EndoscopePosture
GET
nextScopePosture:= m_nextEndoscopePosture;
END_GET
SET
m_nextEndoscopePosture := nextScopePosture;
END_SET
END_PROPERTY

PROPERTY nextScopeType : E_EndoscopePosture
GET
nextScopeType:= m_nextEndoscopeType;
END_GET
SET
m_nextEndoscopeType := nextScopeType;
END_SET
END_PROPERTY

PROPERTY onChipData : REFERENCE TO ST_InstruOnChipData
GET
onChipData ref=m_onChipData;
END_GET
END_PROPERTY

METHOD PROTECTED proGrsapForcepsGripAngleFK : BOOL
VAR_INPUT
	frontAngle:LREAL;
END_VAR
VAR_OUTPUT
	endAngle:LREAL;
	Succeed:BOOL;
END_VAR
VAR
	// prograsp data
	AB :LREAL := 2.8;
	BC:LREAL := 5.26;
	initA:LREAL := 16.6 * g_deg2Rad; 
	initC:LREAL := 8.75*g_deg2Rad;
	
	SIN_C,Angle_Inc_C,Angle_C,Angle_A,Angle_Inc_A:LREAL;
END_VAR
//**************已知：器械前端开合角，求解：末端开合角***************//
// determine prograsp type data
IF InstruType_ProGraspForceps=m_instruType THEN
	AB:=g_proGraspAB;
	BC:=g_proGraspBC;
	initA := g_proGraspInitA;
	initC := g_proGraspInitC;
ELSIF InstruType_ForceBipolar=m_instruType THEN
	AB:=g_proGrasp2AB;
	BC:=g_proGrasp2BC;
	initA := g_proGrasp2InitA;
	initC := g_proGrasp2InitC;
END_IF

Angle_Inc_A:=frontAngle/2;
Angle_A:=initA+Angle_Inc_A;
Angle_A := LIMIT(0.0, Angle_A, pi);

SIN_C:=limit(-1, AB*SIN(Angle_A)/BC, 1);
Angle_C:=ASIN(SIN_C);

Angle_Inc_C:=Angle_C-initC;
endAngle:=Angle_Inc_C*2;
END_METHOD

METHOD PROTECTED proGrsapForcepsGripAngleIK : BOOL
VAR_INPUT
	endAngle:LREAL;
END_VAR
VAR_OUTPUT
	frontAngle:LREAL;
	Succeed:BOOL;
END_VAR
VAR
	AB :LREAL := 2.8;
	BC:LREAL := 5.26;
	initA:LREAL := 16.6 * g_deg2Rad; 
	initC:LREAL := 8.75*g_deg2Rad;
	Angle_Inc_C,Angle_C,SIN_A,Angle_A,Angle_Inc_A:LREAL;
END_VAR
//***************已知：器械末端开合角，求解：前端开合角********************//
// determine prograsp type data
IF InstruType_ProGraspForceps=m_instruType THEN
	AB:=g_proGraspAB;
	BC:=g_proGraspBC;
	initA := g_proGraspInitA;
	initC := g_proGraspInitC;
ELSIF InstruType_ForceBipolar=m_instruType THEN
	AB:=g_proGrasp2AB;
	BC:=g_proGrasp2BC;
	initA := g_proGrasp2InitA;
	initC := g_proGrasp2InitC;
END_IF

Angle_Inc_C:=endAngle/2;
Angle_C:=initC+Angle_Inc_C;
Angle_C := LIMIT(0, Angle_C, pi);

SIN_A:=limit(-1, BC*SIN(Angle_C)/AB, 1);
Angle_A:=ASIN(SIN_A);

Angle_Inc_A:=Angle_A-initA;
frontAngle:=Angle_Inc_A*2;
END_METHOD

METHOD PUBLIC readParameters : BOOL
VAR_INPUT
	startFlag :BOOL;
END_VAR

VAR
	paramIdx :INT;
	endoscopeData:UINT;
END_VAR
// TODO: read m_kinematic parameters from chip 
//Take the rising edge of the read signal
m_ReadDelay(IN:= m_Step=10 OR m_Step=2, PT:= m_DealyTime, Q=> , ET=> );//计时器
IF startFlag AND m_curReadTries < m_maxReadTries THEN
	m_Step:=0;
	m_onChipData.m_InstruReadSucceed:=FALSE;
	m_onChipData.m_Error:=FALSE;
	m_onChipData.m_ErrorID:=0;
	m_resetArmLEDFlag :=TRUE;
	
END_IF


CASE m_Step OF
	0:	m_Value:=0;
		m_SdoWrite(sNetId:= m_ArmNetId, nSlaveAddr:= m_JointInstruAddr, nSubIndex:= 0, nIndex:= 16#6098, pSrcBuf:= ADR(m_Value), cbBufLen:= SIZEOF(m_Value), bExecute:= TRUE, );
		IF NOT m_SdoWrite.bBusy THEN
			m_SdoWrite(bExecute:=FALSE);
			m_Step:=2;
		END_IF
			
	2://延时0.5s、防止值还没有返回
		IF m_ReadDelay.Q THEN
			m_Step:=5;
		END_IF
	
	5://向6093发送0x8000  0000---发送读取信号
		m_Value:=16#80000000; 
		m_SdoWrite(sNetId:= m_ArmNetId, nSlaveAddr:= m_JointInstruAddr, nSubIndex:= 0, nIndex:= 16#6093, pSrcBuf:= ADR(m_Value), cbBufLen:= SIZEOF(m_Value), bExecute:= TRUE, );
		IF NOT m_SdoWrite.bBusy THEN
			m_SdoWrite(bExecute:=FALSE);
			m_Step:=10;
		END_IF
		
		
	10://延时0.5s、防止值还没有返回
		IF m_ReadDelay.Q THEN
			m_Step:=20;
		END_IF

		
	20://从6093地址中拿值
		m_SdoRead(sNetId:= m_ArmNetId, nSlaveAddr:= m_JointInstruAddr,	nSubIndex:= 0, nIndex:= 16#6093, pDstBuf:= ADR(m_IDReadResult), cbBufLen:= SIZEOF(m_IDReadResult), bExecute:= TRUE, 	tTimeout:= , bBusy=> , bError=> , nErrId=> , cbRead=> );
		IF NOT m_SdoRead.bBusy THEN
			m_SdoRead(bExecute:=FALSE);
			m_Step:=30;
		END_IF	
		
	
	30://处理器械ID、低16位
		m_IDResult:=UDINT_TO_ULINT(16#0000FFFF AND m_IDReadResult);
		m_Step:=40;
		
		
	40://读取6095、器械序列号
		m_SdoRead(sNetId:= m_ArmNetId, nSlaveAddr:= m_JointInstruAddr,	nSubIndex:= 0, nIndex:= 16#6095, pDstBuf:= ADR(m_SeriesReadResult), cbBufLen:= SIZEOF(m_SeriesReadResult), bExecute:= TRUE, 	tTimeout:= , bBusy=> , bError=> , nErrId=> , cbRead=> );
		IF NOT m_SdoRead.bBusy THEN
			m_SdoRead(bExecute:=FALSE);
			m_Step:=50;
		END_IF	
	50://处理序列号，低30位
		m_onChipData.m_InstruseriesNum:=SHL(m_IDResult,31)+(16#7FFFFFFF AND m_SeriesReadResult);
		m_onChipData.m_InstruID:=LREAL_TO_INT(FLOOR(lr_in:= m_onChipData.m_InstruseriesNum/EXPT(10,9))); //取十进制前三位为器械ID
		IF m_onChipData.m_InstruID = InstruType_Endoscope  THEN
			endoscopeData := LREAL_TO_UINT(FLOOR(lr_in:= m_onChipData.m_InstruseriesNum/EXPT(10,7)));
			endoscopeData := endoscopeData MOD 100;
			IF endoscopeData>= 25 THEN
				m_onChipData.m_InstruID := InstruType_NewEndoscope;
			END_IF
		ELSIF m_onChipData.m_InstruID = InstruType_CENewEndoscope THEN
			m_onChipData.m_InstruID := InstruType_NewEndoscope;
		END_IF
		InstruIDMap();
		m_Step:=60;
		
	60://读取6096---器械零点位置
		m_SdoRead(sNetId:= m_ArmNetId, nSlaveAddr:= m_JointInstruAddr,	nSubIndex:= 0, nIndex:= 16#6096, pDstBuf:= ADR(m_PosReadResult), cbBufLen:= SIZEOF(m_PosReadResult), bExecute:= TRUE, 	tTimeout:= , bBusy=> , bError=> , nErrId=> , cbRead=> );
		IF NOT m_SdoRead.bBusy THEN
			m_SdoRead(bExecute:=FALSE);
			m_Step:=70;
		END_IF	
		
		
	70: //处理位置，L1:0-9位，L2:10-19位，L3:20-29位
		zeroPosDecode(m_PosReadResult, o_q1=>m_onChipData.m_InstruPos[1],o_q2=>m_onChipData.m_InstruPos[2],o_q3=>m_onChipData.m_InstruPos[3]);
		m_onChipData.m_InstruPos[4] := m_jnt4ZeroPos;
		m_onChipData.m_InstruPos[5] := 0;
		
		m_Step:=80;
		
	80://读取器械使用次数 6094
		m_SdoRead(sNetId:= m_ArmNetId, nSlaveAddr:= m_JointInstruAddr,	nSubIndex:= 0, nIndex:= 16#6094, pDstBuf:= ADR(m_UsageReadResult), cbBufLen:= SIZEOF(m_UsageReadResult), bExecute:= TRUE, 	tTimeout:= , bBusy=> , bError=> , nErrId=> , cbRead=> );
		IF NOT m_SdoRead.bBusy THEN
			m_SdoRead(bExecute:=FALSE);
			m_Step:=90;
		END_IF	
		
		
	90://处理器械使用次数读取结果
		m_onChipData.m_InstruusageCounts:=m_UsageReadResult;
		m_InstruUsageToLED:=LIMIT(0,m_UsageReadResult,99);
		m_Step:=100;
		
		
	100://将器械使用次数写入LED
		m_Value:=ULINT_TO_UDINT(16#FFFF AND m_InstruUsageToLED) ;
//		m_SdoWrite(sNetId:= m_ArmNetId, nSlaveAddr:= m_LEDAddr, nSubIndex:= 06, nIndex:= 16#6090, pSrcBuf:= ADR(m_Value), cbBufLen:= SIZEOF(m_Value), bExecute:= TRUE, tTimeout:= , bBusy=> , bError=> , nErrId=> );
		IF NOT m_SdoWrite.bBusy THEN
			m_SdoWrite(bExecute:=FALSE);
			m_Step:=110;
		END_IF
		
	110:
		m_SdoRead(sNetId:= m_ArmNetId, nSlaveAddr:= m_JointInstruAddr,	nSubIndex:= 0, nIndex:= 16#6097, pDstBuf:= ADR(m_purposeReadResult), cbBufLen:= SIZEOF(m_purposeReadResult), bExecute:= TRUE, 	tTimeout:= , bBusy=> , bError=> , nErrId=> , cbRead=> );
		IF NOT m_SdoRead.bBusy THEN
			m_SdoRead(bExecute:=FALSE);
			m_Step:=120;
		END_IF	
		
		
	120:
		m_onChipData.m_InstruPurpose:=SHR(m_purposeReadResult,16) AND 16#7FFF;
		m_onChipData.m_InstruPurposeTime:=m_purposeReadResult AND 16#FFFF;
		m_Step:=130;
	
	130:
		// get insturment typeinfo
		m_onChipData.m_InstruReadSucceed:=checkInstruType();
		
		//结果诊断
		m_onChipData.m_ErrorID:=0;
		IF NOT(m_onChipData.m_InstruReadSucceed) THEN
			m_onChipData.m_Error:=TRUE;
			m_onChipData.m_ErrorID:=1;
			
			IF m_onChipData.m_InstruPurposeTime < m_instruTypeInfo.m_maxUseNum THEN
				m_onChipData.m_InstruPurposeTime:= m_instruTypeInfo.m_maxUseNum;
			END_IF
//		ELSIF SlaveArmControl.m_slaveRobot.m_endoscopeMounted AND m_instruType = InstruType_Endoscope THEN
//			m_onChipData.m_InstruReadSucceed := FALSE;
//			m_onChipData.m_Error:=TRUE;
//			m_onChipData.m_ErrorID:=3;
			
//		ELSIF m_onChipData.m_InstruusageCounts>(m_instruTypeInfo.m_maxUseNum -1) AND m_instruType<>InstruType_Endoscope THEN
//			m_HaveRecord:=InstruSreiesFind(i_NewValue:=m_onChipData.m_InstruseriesNum , i_ArrayData:=GVL_interactUI.g_InstruSeriesRecord );
//			IF m_HaveRecord THEN
//				//
//			ELSE
//				m_onChipData.m_InstruReadSucceed := FALSE; 
//				m_onChipData.m_Error:=TRUE;
//				m_onChipData.m_ErrorID:=2;
//			END_IF
		END_IF
		
		//处理当器械使用次数达到上限后、在同一场手术中还能使用
//		IF m_onChipData.m_InstruReadSucceed AND m_onChipData.m_InstruusageCounts=(m_instruTypeInfo.m_maxUseNum -1) THEN		
//			//TODO: check this part
//			GVL_interactUI.g_InstruSeriesRecord:=InstruIDRecord(i_NewValue:= m_onChipData.m_InstruseriesNum, i_ArrayData:= GVL_interactUI.g_InstruSeriesRecord);
//		END_IF
		
		m_Step :=-1;
		m_curReadTries := m_curReadTries +1;
	
END_CASE
END_METHOD

METHOD PUBLIC readParametersRFID : BOOL
VAR_INPUT
	startFlag :BOOL;
END_VAR

VAR
	paramIdx :INT;
	endoscopeData:UINT;
END_VAR
// TODO: read m_kinematic parameters from chip 
//Take the rising edge of the read signal
m_ReadDelayRFID(IN:= m_StepRFID=10 OR m_StepRFID=2, PT:= m_DealyTime, Q=> , ET=> );//计时器
IF startFlag  THEN
	m_StepRFID:=0;
	m_onChipData.m_InstruReadSucceedRFID:=FALSE;
END_IF


CASE m_StepRFID OF
	0:	m_Value:=1;
		m_SdoWrite(sNetId:= m_ArmNetId, nSlaveAddr:= m_JointInstruAddr, nSubIndex:= 0, nIndex:= 16#6098, pSrcBuf:= ADR(m_Value), cbBufLen:= SIZEOF(m_Value), bExecute:= TRUE, );
		IF NOT m_SdoWrite.bBusy THEN
			m_SdoWrite(bExecute:=FALSE);
			m_StepRFID:=2;
		END_IF
			
	2://延时0.5s、防止值还没有返回
		IF m_ReadDelayRFID.Q THEN
			m_StepRFID:=5;
		END_IF
	
	5://向6093发送0x8000  0000---发送读取信号
		m_Value:=16#80000000; 
		m_SdoWrite(sNetId:= m_ArmNetId, nSlaveAddr:= m_JointInstruAddr, nSubIndex:= 0, nIndex:= 16#6093, pSrcBuf:= ADR(m_Value), cbBufLen:= SIZEOF(m_Value), bExecute:= TRUE, );
		IF NOT m_SdoWrite.bBusy THEN
			m_SdoWrite(bExecute:=FALSE);
			m_StepRFID:=10;
		END_IF
		
		
	10://延时0.5s、防止值还没有返回
		IF m_ReadDelayRFID.Q THEN
			m_StepRFID:=20;
		END_IF

		
	20://从6093地址中拿值
		m_SdoRead(sNetId:= m_ArmNetId, nSlaveAddr:= m_JointInstruAddr,	nSubIndex:= 0, nIndex:= 16#6093, pDstBuf:= ADR(m_IDReadResult), cbBufLen:= SIZEOF(m_IDReadResult), bExecute:= TRUE, 	tTimeout:= , bBusy=> , bError=> , nErrId=> , cbRead=> );
		IF NOT m_SdoRead.bBusy THEN
			m_SdoRead(bExecute:=FALSE);
			m_StepRFID:=30;
		END_IF	
		
	
	30://处理器械ID、低16位
		m_IDResult:=UDINT_TO_ULINT(16#0000FFFF AND m_IDReadResult);
		m_StepRFID:=40;
		
		
	40://读取6095、器械序列号
		m_SdoRead(sNetId:= m_ArmNetId, nSlaveAddr:= m_JointInstruAddr,	nSubIndex:= 0, nIndex:= 16#6095, pDstBuf:= ADR(m_SeriesReadResult), cbBufLen:= SIZEOF(m_SeriesReadResult), bExecute:= TRUE, 	tTimeout:= , bBusy=> , bError=> , nErrId=> , cbRead=> );
		IF NOT m_SdoRead.bBusy THEN
			m_SdoRead(bExecute:=FALSE);
			m_StepRFID:=50;
		END_IF	
	50://处理序列号，低30位
		m_onChipData.m_InstruseriesNumRFID:=SHL(m_IDResult,31)+(16#7FFFFFFF AND m_SeriesReadResult);
		m_onChipData.m_InstruIDFromRFID:=LREAL_TO_INT(FLOOR(lr_in:= m_onChipData.m_InstruseriesNumRFID/EXPT(10,9))); //取十进制前三位为器械ID
		IF m_onChipData.m_InstruIDFromRFID = InstruType_Endoscope THEN
			endoscopeData := LREAL_TO_UINT(FLOOR(lr_in:= m_onChipData.m_InstruseriesNumRFID/EXPT(10,7)));
			endoscopeData := endoscopeData MOD 100;
			IF endoscopeData>= 25 THEN
				m_onChipData.m_InstruIDFromRFID := InstruType_NewEndoscope;
			END_IF
		END_IF
		m_StepRFID:=60;
		
	60://读取6096---器械零点位置
		m_SdoRead(sNetId:= m_ArmNetId, nSlaveAddr:= m_JointInstruAddr,	nSubIndex:= 0, nIndex:= 16#6096, pDstBuf:= ADR(m_PosReadResult), cbBufLen:= SIZEOF(m_PosReadResult), bExecute:= TRUE, 	tTimeout:= , bBusy=> , bError=> , nErrId=> , cbRead=> );
		IF NOT m_SdoRead.bBusy THEN
			m_SdoRead(bExecute:=FALSE);
			m_StepRFID:=70;
		END_IF	
		
		
	70: //处理位置，L1:0-9位，L2:10-19位，L3:20-29位
		zeroPosDecode(m_PosReadResult, o_q1=>m_onChipData.m_InstruPosRFID[1],o_q2=>m_onChipData.m_InstruPosRFID[2],o_q3=>m_onChipData.m_InstruPosRFID[3]);
		m_onChipData.m_InstruPosRFID[4] := m_jnt4ZeroPos;
		m_onChipData.m_InstruPosRFID[5] := 0;
		
		m_StepRFID:=80;
		
	80://读取器械使用次数 6094
		m_SdoRead(sNetId:= m_ArmNetId, nSlaveAddr:= m_JointInstruAddr,	nSubIndex:= 0, nIndex:= 16#6094, pDstBuf:= ADR(m_UsageReadResult), cbBufLen:= SIZEOF(m_UsageReadResult), bExecute:= TRUE, 	tTimeout:= , bBusy=> , bError=> , nErrId=> , cbRead=> );
		IF NOT m_SdoRead.bBusy THEN
			m_SdoRead(bExecute:=FALSE);
			m_StepRFID:=90;
		END_IF	
		
		
	90://处理器械使用次数读取结果
		m_onChipData.m_InstruUsageCountsRFID:=m_UsageReadResult;
		m_StepRFID:=-1;
		m_onChipData.m_InstruReadSucceedRFID:=TRUE;
(*		
	100://将器械使用次数写入LED
		m_Value:=ULINT_TO_UDINT(16#FFFF AND m_InstruUsageToLED) ;
//		m_SdoWrite(sNetId:= m_ArmNetId, nSlaveAddr:= m_LEDAddr, nSubIndex:= 06, nIndex:= 16#6090, pSrcBuf:= ADR(m_Value), cbBufLen:= SIZEOF(m_Value), bExecute:= TRUE, tTimeout:= , bBusy=> , bError=> , nErrId=> );
		IF NOT m_SdoWrite.bBusy THEN
			m_SdoWrite(bExecute:=FALSE);
			m_Step:=110;
		END_IF
		
	110:
		m_SdoRead(sNetId:= m_ArmNetId, nSlaveAddr:= m_JointInstruAddr,	nSubIndex:= 0, nIndex:= 16#6097, pDstBuf:= ADR(m_purposeReadResult), cbBufLen:= SIZEOF(m_purposeReadResult), bExecute:= TRUE, 	tTimeout:= , bBusy=> , bError=> , nErrId=> , cbRead=> );
		IF NOT m_SdoRead.bBusy THEN
			m_SdoRead(bExecute:=FALSE);
			m_Step:=120;
		END_IF	
		
		
	120:
		m_onChipData.m_InstruPurpose:=SHR(m_purposeReadResult,16) AND 16#7FFF;
		m_onChipData.m_InstruPurposeTime:=m_purposeReadResult AND 16#FFFF;
		m_Step:=130;
	
	130:
		// get insturment typeinfo
		m_onChipData.m_InstruReadSucceed:=checkInstruType();
		
		//结果诊断
		m_onChipData.m_ErrorID:=0;
		IF NOT(m_onChipData.m_InstruReadSucceed) THEN
			m_onChipData.m_Error:=TRUE;
			m_onChipData.m_ErrorID:=1;
			
//		ELSIF SlaveArmControl.m_slaveRobot.m_endoscopeMounted AND m_instruType = InstruType_Endoscope THEN
//			m_onChipData.m_InstruReadSucceed := FALSE;
//			m_onChipData.m_Error:=TRUE;
//			m_onChipData.m_ErrorID:=3;
			
//		ELSIF m_onChipData.m_InstruusageCounts>(m_instruTypeInfo.m_maxUseNum -1) AND m_instruType<>InstruType_Endoscope THEN
//			m_HaveRecord:=InstruSreiesFind(i_NewValue:=m_onChipData.m_InstruseriesNum , i_ArrayData:=GVL_interactUI.g_InstruSeriesRecord );
//			IF m_HaveRecord THEN
//				//
//			ELSE
//				m_onChipData.m_InstruReadSucceed := FALSE; 
//				m_onChipData.m_Error:=TRUE;
//				m_onChipData.m_ErrorID:=2;
//			END_IF
		END_IF
		
		//处理当器械使用次数达到上限后、在同一场手术中还能使用
//		IF m_onChipData.m_InstruReadSucceed AND m_onChipData.m_InstruusageCounts=(m_instruTypeInfo.m_maxUseNum -1) THEN		
//			//TODO: check this part
//			GVL_interactUI.g_InstruSeriesRecord:=InstruIDRecord(i_NewValue:= m_onChipData.m_InstruseriesNum, i_ArrayData:= GVL_interactUI.g_InstruSeriesRecord);
//		END_IF
		
		m_Step :=-1;
		m_curReadTries := m_curReadTries +1;
	*)
END_CASE
END_METHOD

METHOD PUBLIC reset : BOOL
VAR_INPUT
END_VAR
VAR
	i:INT;
END_VAR
m_Step := -1;
m_StepRFID:=-1;
m_curReadTries := 0;
m_onChipData.m_InstruID := 0;
m_onChipData.m_InstruseriesNum :=0;
m_onChipData.m_Error:=FALSE;
m_onChipData.m_ErrorID:=0;
m_onChipData.m_InstruReadSucceed:=FALSE;
m_instruType:=InstruType_UNKNOWM;

m_instruTypeInfo.m_instruNameCH := "";
m_onChipData.m_InstruIDFromRFID := 0;
m_onChipData.m_InstruseriesNumRFID :=0;
m_onChipData.m_InstruReadSucceedRFID:=FALSE;
FOR i:= 4 TO 8 BY 1 DO
	m_jntPosOffset[i]:=0;
END_FOR

// init joint motion range
FOR i:=1 TO 3 DO
	m_wristMinDHJntPos[i]:=GVL_SlaveMotorParameters.g_minDHJntPos[i+3];
	m_wristMaxDHJntPos[i]:=GVL_SlaveMotorParameters.g_maxDHJntPos[i+3];
END_FOR

// reset endoscope type and posture
m_curEndoscopeType :=EndoScopeType_30;
m_nextEndoscopeType :=EndoScopeType_30;
m_curEndoscopePosture :=EndoscopePosture_HeadDown;
m_nextEndoscopePosture :=EndoscopePosture_HeadDown;

//arm LED reset
IF m_resetArmLEDFlag THEN
	m_Value:=0 ;
//	m_SdoWrite(sNetId:= m_ArmNetId, nSlaveAddr:= m_LEDAddr, nSubIndex:= 06, nIndex:= 16#6090, pSrcBuf:= ADR(m_Value), cbBufLen:= SIZEOF(m_Value), bExecute:= TRUE, tTimeout:= , bBusy=> , bError=> , nErrId=> );
END_IF
IF NOT m_SdoWrite.bBusy THEN
	m_SdoWrite(bExecute:=FALSE);
	m_resetArmLEDFlag := FALSE;
END_IF

//Reset zero pos
FOR i:=1 TO 5 DO
	m_onChipData.m_InstruPos[i]:=0;
	m_onChipData.m_InstruPosRFID[i]:=0;
END_FOR
onChipData.m_InstruusageCounts:=0;
onChipData.m_InstruPurpose:=0;
onChipData.m_InstruPurposeTime:=0;
onChipData.m_InstruUsageCountsRFID:=0;
END_METHOD

PROPERTY resetArmLED : BOOL
SET
m_resetArmLEDFlag := resetArmLED;
END_SET
END_PROPERTY

METHOD ultrasoundKnifeGripAngleFK : LREAL
VAR_INPUT
	// motor joint position of slave arm
	i_jntPos :LREAL;
END_VAR

VAR
	m_jntPos : LREAL;
END_VAR
m_jntPos := i_jntPos;

m_jntPos := LIMIT (-20*g_deg2Rad,m_jntPos,70*g_deg2Rad);

ultrasoundKnifeGripAngleFK := ASIN((m_jntPos*g_uknifeMotorLead * g_uknifeLeverRatio/(2*pi) -  g_uknifeGripTravel * SIN(g_uknifeGripDividAngle))/g_uknifeGripTravel)+g_uknifeGripDividAngle;
END_METHOD

METHOD ultrasoundKnifeGripAngleIK : LREAL
VAR_INPUT
	// gripper angle
	i_gripAngle :LREAL;
END_VAR

VAR
	m_gripAngle : LREAL;
END_VAR
m_gripAngle := i_gripAngle;

ultrasoundKnifeGripAngleIK := (g_uknifeGripTravel * (SIN(g_uknifeGripDividAngle) - SIN(g_uknifeGripDividAngle - m_gripAngle))/(g_uknifeMotorLead*g_uknifeLeverRatio/(2*pi)));
END_METHOD

METHOD writeNumOfUseToChip : BOOL
VAR_INPUT
	startFlag :BOOL;
	i_useNumFromUI :UINT;
END_VAR
writeNumOfUseToChip := FALSE;
m_writeLDP(CLK:= startFlag, Q=> );
m_ReadNumDelay(IN:= m_useNumStep = 10, PT:= m_DealyTime, Q=> , ET=> );
IF m_writeLDP.Q THEN
	m_useNumStep:=0;
END_IF

CASE m_useNumStep OF
	0: 
		m_Value:=16#80000000; 
		m_SdoWrite(sNetId:= m_ArmNetId, nSlaveAddr:= m_JointInstruAddr, nSubIndex:= 0, nIndex:= 16#6094, pSrcBuf:= ADR(m_Value), cbBufLen:= SIZEOF(m_Value), bExecute:= TRUE, );
		IF NOT m_SdoWrite.bBusy THEN
			m_SdoWrite(bExecute:=FALSE);
			m_useNumStep:=10;
		END_IF
	
	10:
		IF m_ReadNumDelay.Q THEN
			m_useNumStep:=20;
		END_IF
		
	20:
		m_SdoRead(sNetId:= m_ArmNetId, nSlaveAddr:= m_JointInstruAddr,	nSubIndex:= 0, nIndex:= 16#6094, pDstBuf:= ADR(m_useNumReadResult), cbBufLen:= SIZEOF(m_useNumReadResult), bExecute:= TRUE, 	tTimeout:= , bBusy=> , bError=> , nErrId=> , cbRead=> );
		IF NOT m_SdoRead.bBusy THEN
			m_SdoRead(bExecute:=FALSE);
			m_useNumStep:=30;
		END_IF
		
	30://Verify the actual usage count and the usage count given by the UI
		IF m_useNumReadResult = i_useNumFromUI THEN
			m_useNumSendToLED := LIMIT(0, m_useNumReadResult, 99);
			m_useNumStep:=40;
		ELSE
			m_useNumStep:=50;
		END_IF
		
	40: 
		m_Value:=ULINT_TO_UDINT( m_useNumSendToLED) ;
//		m_SdoWrite(sNetId:= m_ArmNetId, nSlaveAddr:= m_LEDAddr, nSubIndex:= 06, nIndex:= 16#6090, pSrcBuf:= ADR(m_Value), cbBufLen:= SIZEOF(m_Value), bExecute:= TRUE, tTimeout:= , bBusy=> , bError=> , nErrId=> );
		IF NOT m_SdoWrite.bBusy THEN
			m_SdoWrite(bExecute:=FALSE);
			m_onChipData.m_InstruUsageCounts:=m_useNumReadResult;
			writeNumOfUseToChip := TRUE;
			m_useNumStep:=-1;
		END_IF
		
END_CASE
END_METHOD

METHOD writePurpose : BOOL
VAR
	instruMaxUsed : UINT;
END_VAR
IF InstruType_Endoscope=m_instruType OR InstruType_NewEndoscope=m_instruType THEN
	m_purposeMode:=GVL_InstruTestUIVars.g_writePurposeNum+10;
ELSIF InstruType_UltrasoundKnifeS=m_instruType OR InstruType_UltrasoundKnifeU=m_instruType THEN 
	m_purposeMode:=GVL_InstruTestUIVars.g_writePurposeNum+20;
ELSE
	m_purposeMode:=GVL_InstruTestUIVars.g_writePurposeNum;
END_IF
IF m_instruTypeInfo.m_maxUseNum <> 0 THEN
	instruMaxUsed := m_instruTypeInfo.m_maxUseNum;
ELSE
	instruMaxUsed := 10;
END_IF

CASE m_purposeMode OF
	1: m_Value:=instruMaxUsed OR 16#10000; 
	2: m_Value:=16#3E7 OR 16#20000; 
	3: m_Value:=instruMaxUsed OR 16#30000; 
	4: m_Value:=16#1E OR 16#40000; 
	11: m_Value:=16#64 OR 16#10000; 
	12: m_Value:=16#3E7 OR 16#20000; 
	13: m_Value:=16#64 OR 16#30000; 
	14: m_Value:=16#64 OR 16#40000; 
ELSE
	RETURN;
END_CASE
m_Value:=m_Value OR 16#80000000; 
m_SdoWrite(sNetId:= m_ArmNetId, nSlaveAddr:= m_JointInstruAddr, nSubIndex:= 0, nIndex:= 16#6097, pSrcBuf:= ADR(m_Value), cbBufLen:= SIZEOF(m_Value), bExecute:= TRUE, );
IF NOT m_SdoWrite.bBusy THEN
	m_SdoWrite(bExecute:=FALSE);
	writePurpose := 1;
END_IF
END_METHOD

METHOD writeSNToChip : BOOL
VAR_INPUT
	newSNNum : ULINT;
END_VAR
VAR
	
END_VAR
// TODO
m_fbTon_Step[1](IN:=m_SDOStep=5 , PT:= T#1S, Q=> , ET=> );
m_fbTon_Step[2](IN:=m_SDOStep=15 , PT:= T#1S, Q=> , ET=> );
CASE m_SDOStep OF
	0: 
	  value:=(newSNNum AND 16#7FFFFFFF)OR 16#80000000;
	  m_SDOStep:=5;
	5:	
	  m_SdoWrite(sNetId:= m_ArmNetId, nSlaveAddr:= m_JointInstruAddr, nSubIndex:= 0, nIndex:= 16#6095, pSrcBuf:= ADR(value), cbBufLen:= SIZEOF(value), bExecute:= TRUE, );
	  IF NOT m_SdoWrite.bBusy AND m_fbTon_Step[1].Q THEN
		  m_SdoWrite(bExecute:=FALSE);
		  m_SDOStep:=10;
	  END_IF
	10:
	  value:=SHR(newSNNum,31)OR 16#10000;
	  m_SDOStep:=15;
	15: 
	  m_SdoWrite(sNetId:= m_ArmNetId, nSlaveAddr:= m_JointInstruAddr, nSubIndex:= 0, nIndex:= 16#6093, pSrcBuf:= ADR(value), cbBufLen:= SIZEOF(value), bExecute:= TRUE, );
	  IF NOT m_SdoWrite.bBusy AND m_fbTon_Step[2].Q THEN
		  m_SdoWrite(bExecute:=FALSE);
		  writeSNToChip:=TRUE;
		  m_SDOStep:=0;
	  END_IF
END_CASE
END_METHOD

METHOD PUBLIC writeZeroPosToChip : BOOL
VAR_INPUT
	i_q1:LREAL;
	i_q2:LREAL;
	i_q3:LREAL;
END_VAR
zeroPosCode(i_q1,i_q2,i_q3, o_code=>m_zeroPosCode);

writeZeroPosToChip:=FALSE;
m_SdoWrite(sNetId:= m_ArmNetId, nSlaveAddr:= m_JointInstruAddr, nSubIndex:= 0, nIndex:= 16#6096, pSrcBuf:= ADR(m_zeroPosCode), cbBufLen:= SIZEOF(m_zeroPosCode), bExecute:= TRUE, );
IF NOT m_SdoWrite.bBusy THEN
	m_SdoWrite(bExecute:=FALSE);
	writeZeroPosToChip:=TRUE;
END_IF
END_METHOD

// code instrument joints(4/5/6) zero position as a UDINT
// joint1 : bit 21-30; joint2: bit 11-20; joint3: bit1-10
// zeroPos: [0, 2pi]; code:[0-3sFF]
METHOD PROTECTED zeroPosCode : BOOL
VAR_INPUT
	i_q1:LREAL;
	i_q2:LREAL;
	i_q3:LREAL;
END_VAR
VAR_OUTPUT
	o_code:UDINT;
END_VAR
VAR
	posCode:UDINT;
END_VAR
// highest bit set to 1
o_code:=2;

// joint1
posCode := LREAL_TO_UDINT(16#3FF * LIMIT(0,i_q1/g_2pi,1));
o_code := SHL(o_code, 10);
o_code := o_code OR posCode;

// joint2
posCode := LREAL_TO_UDINT(16#3FF * LIMIT(0,i_q2/g_2pi,1));
o_code := SHL(o_code, 10);
o_code := o_code OR posCode;

// joint3
posCode := LREAL_TO_UDINT(16#3FF * LIMIT(0,i_q3/g_2pi,1));
o_code := SHL(o_code, 10);
o_code := o_code OR posCode;
END_METHOD

// decode instrument joints(4/5/6) zero position from a UDINT
// joint1 : bit 21-30; joint2: bit 11-20; joint4: bit1-10
// zeroPos: [0, 2pi]; code:[0-2FF]
METHOD PROTECTED zeroPosDecode : BOOL
VAR_INPUT
	i_posCode :UDINT;
END_VAR
VAR_OUTPUT
	o_q1:LREAL;
	o_q2:LREAL;
	o_q3:LREAL;
END_VAR
VAR
	posCode:UDINT;
END_VAR
// joint3
posCode := i_posCode AND 16#3FF;
o_q3 := g_2pi *  posCode/16#3FF;

// joint2
i_posCode := SHR(i_posCode, 10);
posCode := i_posCode AND 16#3FF;
o_q2 := g_2pi *  posCode/16#3FF;

// joint1
i_posCode := SHR(i_posCode, 10);
posCode := i_posCode AND 16#3FF;
o_q1 := g_2pi *  posCode/16#3FF;
END_METHOD

END_FUNCTION_BLOCK

// ---- FBs_Auxiliary/FB_initMotorPID.TcPOU
FUNCTION_BLOCK FB_initMotorPID
VAR_INPUT
END_VAR
VAR_OUTPUT
END_VAR
VAR
	m_SdoWrite:FB_EcCoESdoWrite;
	m_SdoRead:FB_EcCoESdoRead;
	m_step:INT;
	m_armIdx :INT;
	m_jntIdx :INT;
	m_curjntIdx: INT;
	//IP of operating arm
	m_armNetId:T_AmsNetId; 	
	
	//Joint port number
	m_jointPortAddr:ARRAY[1..g_sJntNum] OF UINT ;
	m_Value	:UDINT;
	m_number:INT;
	m_motorPID:ARRAY[1..g_sJntNum,1..6] OF INT;
	m_ton:TON;
	m_readMotorPID:ARRAY[1..g_sJntNum,1..6] OF INT;
	m_clearReadMotorPID:ARRAY[1..g_sJntNum,1..6] OF INT;
	m_motorErrNum:INT;
	m_isFinished:INT;
	m_initPID:BOOL:=FALSE;
	m_stepRun:INT;
	m_armNum:INT;
	m_initFinishPID:ARRAY[1..g_sArmNum] OF BOOL;
	m_robotMotorRunMid:BOOL;
	m_errNum:INT;
	m_errStop:BOOL;
END_VAR

METHOD armMotorRun : BOOL
VAR_INPUT
END_VAR
VAR
	i:INT;
	j:INT;
END_VAR
m_ton(IN:= m_step = 10, PT:= T#100MS, Q=> , ET=> );
CASE m_step OF
	0: ;
	2:
		armMotorRun:=FALSE;
		m_Step:=5;
	5://Write
		m_Value:=INT_TO_UDINT(m_motorPID[m_curjntIdx,m_number] );
		m_SdoWrite(sNetId:= m_ArmNetId, nSlaveAddr:= m_jointPortAddr[m_curjntIdx], nSubIndex:=INT_TO_BYTE( m_number), nIndex:= 16#6090, pSrcBuf:= ADR(m_Value), cbBufLen:= SIZEOF(m_Value), bExecute:= TRUE, tTimeout:= , bBusy=> , bError=> , nErrId=> );
		IF NOT m_SdoWrite.bBusy THEN
			m_SdoWrite(bExecute:=FALSE);
			m_Step:=10;
		END_IF
	10:
 		IF m_ton.Q THEN
			m_step:=15;
		END_IF
	15:
		m_number:=m_number+1;
		m_step:=5;
		IF m_number=6+1 THEN
			m_number:=1;
			m_curjntIdx:=m_curjntIdx+1;
		END_IF
		IF m_curjntIdx=m_jntIdx+1 THEN
			m_number:=1;
			m_curjntIdx:=1;
			m_step:=20;
			m_Value:=0;
		END_IF
	20://Read	
		m_SdoRead(sNetId:= m_ArmNetId, nSlaveAddr:= m_jointPortAddr[m_curjntIdx],	nSubIndex:= INT_TO_BYTE( m_number), nIndex:= 16#6090, pDstBuf:= ADR(m_Value), cbBufLen:= SIZEOF(m_Value), bExecute:= TRUE, 	tTimeout:= , bBusy=> , bError=> , nErrId=> , cbRead=> );
		IF NOT m_SdoRead.bBusy THEN
			m_SdoRead(bExecute:=FALSE);
			m_Step:=25;
		END_IF	
	25:
 		m_readMotorPID[m_curjntIdx,m_number]:=UDINT_TO_INT(m_Value);
		m_Step:=30;
	30:
		m_number:=m_number+1;
		m_step:=20;
		m_Value:=0;
		IF m_number=6+1 THEN
			m_number:=1;
			m_curjntIdx:=m_curjntIdx+1;
		END_IF
		IF m_curjntIdx=m_jntIdx+1 THEN
			m_step:=40;
			m_errStop:=FALSE;
		END_IF
	40:
		FOR i:=1 TO m_jntIdx BY 1 DO
			FOR j:=1 TO 6 BY 1 DO
				IF NOT m_errStop THEN
					IF m_readMotorPID[i,j]<=1.2*m_motorPID[i,j] AND m_readMotorPID[i,j]>=0.8*m_motorPID[i,j]AND m_readMotorPID[i,j]<>m_motorPID[i,j] THEN
						m_motorErrNum:=i;
					END_IF
					IF m_readMotorPID[i,j]>1.2*m_motorPID[i,j] OR m_readMotorPID[i,j]<0.8*m_motorPID[i,j]THEN
						m_motorErrNum:=i*10;
						m_errStop:=TRUE;
					END_IF
				END_IF
			END_FOR
		END_FOR
		m_step:=50;
	50:
		IF m_motorErrNum=0 THEN
			armMotorRun:=TRUE;
		ELSE
			armMotorRun:=FALSE;
		END_IF
		m_step:=0;
END_CASE
END_METHOD

METHOD init : BOOL
VAR_INPUT
	i_armIdx :INT;
END_VAR
VAR
	i:INT;
END_VAR
m_step:=2;
m_armIdx:=i_armIdx;
m_jntIdx:=g_sJntNum;
m_curjntIdx:=1;
m_number:=1;
m_motorErrNum:=0;
m_armNetId:=GVL_SlaveJointEncoderCaliData.g_slaveArmNetID[m_armIdx];
FOR i:=1 TO m_jntIdx BY 1 DO
	m_jointPortAddr[i]:=GVL_SlaveJointEncoderCaliData.g_slaveJointNetPort[m_armIdx,i];
END_FOR

m_motorPID:=GVL_SlaveMotorParameters.g_motorPID;

m_readMotorPID:=m_clearReadMotorPID;
END_METHOD

METHOD robotMotorRun : BOOL
VAR_INPUT
END_VAR
VAR
  i:INT;
END_VAR
//init motor pid
IF m_initPID=0 THEN
	m_stepRun:=5;
	m_armNum:=1;
	m_initPID:=1;
	m_errNum:=0;
	robotMotorRun:=FALSE;
	m_robotMotorRunMid:=FALSE;
	m_isFinished:=5;
END_IF

